// TwinCAT 3 PLC project PRG_Test_Base
// ProgramVersion: 3.1.4024.0
// libraries:
//   B_Base, * (RafalOS)
//   B_Base_HMI_Connector, * (RafalOS)
//   Tc2_Standard, * (Beckhoff Automation GmbH)
//   Tc2_System, * (Beckhoff Automation GmbH)
//   Tc3_Module, * (Beckhoff Automation GmbH)
//   TcUnit, * (www.tcunit.org)
// project tree:
//   GVLs/ GVL.TcGVL, GVL_Variable.TcGVL, GVL_VariableHMI.TcGVL
//   / PlcTask.TcTTO (not stored)
//   POUs/A0_BaseFB/Command/ FB_CommandChild.TcPOU, FB_CommandTest.TcPOU, FB_Impulstest.TcPOU (not stored)
//   POUs/A0_BaseFB/Time/ FB_BaseTimeTest.TcPOU (not stored)
//   POUs/A2_logger/ FB_LoggerTest.TcPOU
//   POUs/A4_Component/ FB_Component.TcPOU, FB_Component_HMI.TcPOU, ITF_Component.TcIO, ITF_Component_HMI.TcIO, ITF_Component_HMI_Connector.TcIO, ITF_Component_HMI_Init.TcIO (not stored), ST_Component_HMI.TcDUT, ST_Component_HMI_Link.TcDUT (not stored)
//   POUs/A5_ControlElement/ FB_ControlElement.TcPOU, FB_ControlElement_HMI.TcPOU, ITF_ControlElement.TcIO, ITF_ControlElement_HMI.TcIO, ITF_ControlElement_HMI_Connector.TcIO, ITF_ControlElement_HMI_Init.TcIO, ST_ControlElement_HMI.TcDUT, ST_ControlElement_HMI_Link.TcDUT
//   POUs/A5_ControlElement_1/ FB_ControlElement_1.TcPOU (not stored), FB_ControlElement_HMI_1.TcPOU (not stored), ITF_ControlElement_1.TcIO, ITF_ControlElement_HMI_1.TcIO (not stored), ITF_ControlElement_HMI_Connector_1.TcIO, ITF_ControlElement_HMI_Init_1.TcIO, ST_ControlElement_HMI_1.TcDUT, ST_ControlElement_HMI_Link_1.TcDUT
//   POUs/A6_GroupElement/ FB_GroupElement.TcPOU, FB_GroupElement_HMI.TcPOU, ITF_GroupElement.TcIO, ITF_GroupElement_HMI.TcIO, ITF_GroupElement_HMI_Connector.TcIO (not stored), ITF_GroupElement_HMI_Init.TcIO, ST_GroupElement_HMI.TcDUT, ST_GroupElement_HMI_Link.TcDUT
//   POUs/A7_TopElement/ FB_TopElement.TcPOU, FB_TopElement_HMI.TcPOU, ITF_TopElement.TcIO, ITF_TopElement_HMI.TcIO, ITF_TopElement_HMI_Connector.TcIO (not stored), ITF_TopElement_HMI_Init.TcIO (not stored), ST_TopElement_HMI.TcDUT, ST_TopElement_HMI_Link.TcDUT
//   POUs/A8_CommunicatorTest/ FB_CommunicatorClient.TcPOU
//   POUs/ FB_ItemTest.TcPOU
//   TESTs/ PRG_Test.TcPOU
// real-time tasks:
//   TASK PlcTask: cycle T#10ms, priority 20, ADS port 350

// ---- POUs/A4_Component/ST_Component_HMI.TcDUT
TYPE ST_Component_HMI EXTENDS ST_BaseComponent_HMI :
STRUCT
	
END_STRUCT
END_TYPE

// ---- POUs/A5_ControlElement/ST_ControlElement_HMI.TcDUT
TYPE ST_ControlElement_HMI :
STRUCT
	bZmiennaControlElement		: BOOL;
	
END_STRUCT
END_TYPE

// ---- POUs/A5_ControlElement/ST_ControlElement_HMI_Link.TcDUT
TYPE ST_ControlElement_HMI_Link EXTENDS ST_BaseControlElement_HMI_Link :
STRUCT
	stControlElement			: ST_ControlElement_HMI;
END_STRUCT
END_TYPE

// ---- POUs/A5_ControlElement_1/ST_ControlElement_HMI_1.TcDUT
TYPE ST_ControlElement_HMI_1 :
STRUCT
	bZmiennaControlElement_1		: BOOL;
	
END_STRUCT
END_TYPE

// ---- POUs/A5_ControlElement_1/ST_ControlElement_HMI_Link_1.TcDUT
TYPE ST_ControlElement_HMI_Link_1 EXTENDS ST_BaseControlElement_HMI_Link :
STRUCT
	stControlElement			: ST_ControlElement_HMI_1;
	
	stComponent1				: ST_Component_HMI_Link;
	stComponent2				: ST_Component_HMI_Link;
	
END_STRUCT
END_TYPE

// ---- POUs/A6_GroupElement/ST_GroupElement_HMI.TcDUT
TYPE ST_GroupElement_HMI :
STRUCT
	bZmiennaGroupElement	: BOOL;
	
END_STRUCT
END_TYPE

// ---- POUs/A6_GroupElement/ST_GroupElement_HMI_Link.TcDUT
TYPE ST_GroupElement_HMI_Link EXTENDS ST_BaseGroupElement_HMI_Link :
STRUCT
	stGroupElement			: ST_GroupElement_HMI;
END_STRUCT
END_TYPE

// ---- POUs/A7_TopElement/ST_TopElement_HMI.TcDUT
TYPE ST_TopElement_HMI :
STRUCT
	bZmiennaTopElement			: BOOL;
	
END_STRUCT
END_TYPE

// ---- POUs/A7_TopElement/ST_TopElement_HMI_Link.TcDUT
TYPE ST_TopElement_HMI_Link EXTENDS ST_BaseTopElement_HMI_Link :
STRUCT
	stTopElement			: ST_TopElement_HMI;

	stControlElement1		: ST_ControlElement_HMI_Link;
	stControlElement2		: ST_ControlElement_HMI_Link;
	stGroupElement1			: ST_GroupElement_HMI_Link;
	stComponent1			: ST_Component_HMI_Link;
	stComponent2			: ST_Component_HMI_Link;
	stComponent3			: ST_Component_HMI_Link;
END_STRUCT
END_TYPE

// ---- GVLs/GVL.TcGVL
{attribute 'qualified_only'}
VAR_GLOBAL
	fbMyTime				: FB_BaseTime;
	fbMyLocation			: FB_BaseLocation;
	fbLogger				: FB_BaseLogger;
	fbSS1					: FB_BaseFlag;
	fbSTO					: FB_BaseFlag;
	
	fbCommandEasy			: FB_BaseCommand;
	fbCommand				: FB_CommandChild;
	
	fbImpuls				: FB_BaseImpulse;
	
	fbCommunicator			: FB_BaseCommunicator;
	
	fbRecipe				: FB_BaseRecipe;
	fbCreatingTemplate1		: FB_CreateTepletate1;
	fbCreatingTemplate2		: FB_CreateTepletate2;
	
	stCommonData			: ST_BaseCommonData;
	
	stTopElementData		: ST_TopElement_HMI_Link;
	
	
END_VAR

// ---- GVLs/GVL_Variable.TcGVL
{attribute 'qualified_only'}
VAR_GLOBAL
	fbBasetest					: FB_Base;
	
	fbPB1_Wyk1_K1				: FB_Component;
	fbPB1_Wyk1_K2				: FB_Component;
	fbPB1_Wyk1					: FB_ControlElement (fbPB1_Wyk1_K1, fbPB1_Wyk1_K2);
	
	fbPB1_Wyk2_K1				: FB_Component;
	fbPB1_Wyk2_K2				: FB_Component;
	fbPB1_Wyk2					: FB_ControlElement_1 (fbPB1_Wyk2_K1, fbPB1_Wyk2_K2);

	fbPB1_ZL1_Wyk1_K1			: FB_Component;
	fbPB1_ZL1_Wyk1_K2			: FB_Component;
	fbPB1_ZL1_Wyk1				: FB_ControlElement (fbPB1_ZL1_Wyk1_K1, fbPB1_ZL1_Wyk1_K2);
	fbPB1_ZL1_Wyk2_K1			: FB_Component;
	fbPB1_ZL1_Wyk2_K2			: FB_Component;
	fbPB1_ZL1_Wyk2				: FB_ControlElement (fbPB1_ZL1_Wyk2_K1, fbPB1_ZL1_Wyk2_K2);
	fbPB1_ZL1_K1				: FB_Component;
	fbPB1_ZL1_K2				: FB_Component;
	fbPB1_ZL1					: FB_GroupElement (fbPB1_ZL1_Wyk1, fbPB1_ZL1_Wyk2, fbPB1_ZL1_K1, fbPB1_ZL1_K2);
	
	fbPB1_K1					: FB_Component;
	fbPB1_K2					: FB_Component;
	fbPB1_K3					: FB_Component;
	
	fbPB1						: FB_TopElement (fbPB1_Wyk1, fbPB1_Wyk2, fbPB1_ZL1, fbPB1_K1, fbPB1_K2, fbPB1_K3);
	
END_VAR

// ---- GVLs/GVL_VariableHMI.TcGVL
{attribute 'qualified_only'}
VAR_GLOBAL
//	fbComponentHMI_1			: FB_Component_HMI (itfBaseLoggerConnector := GVL.fbLogger, itfComponentConnector := GVL_Variable.fbComponent_1);
//	fbControlrElementHMI_1		: FB_ControlElement_HMI (itfBaseLoggerConnector := GVL.fbLogger, itfControlElementConnector := GVL_Variable.fbControlElement_1);
//	fbGroupElementHMI_1			: FB_GroupElement_HMI (itfBaseLoggerConnector := GVL.fbLogger, itfGroupelementConnector := GVL_Variable.fbGroupElement_1);
//	fbTopElementHMI_1			: FB_TopElement_HMI (itfBaseLoggerConnector := GVL.fbLogger, itfTopElementConnector := GVL_Variable.fbTopElement_1);
//
//	fbComponentHMI_1_L			: FB_Component_HMI (itfBaseLoggerConnector := GVL.fbLogger, itfComponentConnector := GVL_Variable.fbComponent_1_L);
//	fbComponentHMI_2_L			: FB_Component_HMI (itfBaseLoggerConnector := GVL.fbLogger, itfComponentConnector := GVL_Variable.fbComponent_2_L);
//	fbComponentHMI_3_L			: FB_Component_HMI (itfBaseLoggerConnector := GVL.fbLogger, itfComponentConnector := GVL_Variable.fbComponent_3_L);

	
END_VAR

// ---- POUs/A4_Component/ITF_Component.TcIO
INTERFACE ITF_Component EXTENDS ITF_BaseComponent

END_INTERFACE

// ---- POUs/A4_Component/ITF_Component_HMI.TcIO
INTERFACE ITF_Component_HMI

METHOD LinkComponentData : BOOL
VAR_INPUT
	stData					: REFERENCE TO ST_Component_HMI_Link;
END_VAR
END_METHOD

END_INTERFACE

// ---- POUs/A4_Component/ITF_Component_HMI_Connector.TcIO
INTERFACE ITF_Component_HMI_Connector EXTENDS ITF_BaseComponent_HMI_Connector

END_INTERFACE

// ---- POUs/A5_ControlElement/ITF_ControlElement.TcIO
INTERFACE ITF_ControlElement

END_INTERFACE

// ---- POUs/A5_ControlElement/ITF_ControlElement_HMI.TcIO
INTERFACE ITF_ControlElement_HMI EXTENDS ITF_BaseComponent_HMI

METHOD LinkControlElementData : BOOL
VAR_INPUT
	stData				: REFERENCE TO ST_ControlElement_HMI_Link;
END_VAR
END_METHOD

END_INTERFACE

// ---- POUs/A5_ControlElement/ITF_ControlElement_HMI_Connector.TcIO
INTERFACE ITF_ControlElement_HMI_Connector EXTENDS ITF_BaseControlElement_HMI_Connector

END_INTERFACE

// ---- POUs/A5_ControlElement/ITF_ControlElement_HMI_Init.TcIO
INTERFACE ITF_ControlElement_HMI_Init EXTENDS ITF_BaseControlElement, ITF_ControlElement_HMI_Connector

END_INTERFACE

// ---- POUs/A5_ControlElement_1/ITF_ControlElement_1.TcIO
INTERFACE ITF_ControlElement_1 EXTENDS ITF_BaseControlElement

END_INTERFACE

// ---- POUs/A5_ControlElement_1/ITF_ControlElement_HMI_Connector_1.TcIO
INTERFACE ITF_ControlElement_HMI_Connector_1 EXTENDS ITF_BaseControlElement_HMI_Connector

END_INTERFACE

// ---- POUs/A5_ControlElement_1/ITF_ControlElement_HMI_Init_1.TcIO
INTERFACE ITF_ControlElement_HMI_Init_1 EXTENDS ITF_BaseControlElement, ITF_ControlElement_HMI_Connector_1

END_INTERFACE

// ---- POUs/A6_GroupElement/ITF_GroupElement.TcIO
INTERFACE ITF_GroupElement EXTENDS ITF_BaseGroupElement

END_INTERFACE

// ---- POUs/A6_GroupElement/ITF_GroupElement_HMI.TcIO
INTERFACE ITF_GroupElement_HMI EXTENDS ITF_BaseGroupElement_HMI

METHOD LinkGroupelementData : BOOL
VAR_INPUT
	stData					: REFERENCE TO ST_GroupElement_HMI_Link;
END_VAR
END_METHOD

END_INTERFACE

// ---- POUs/A6_GroupElement/ITF_GroupElement_HMI_Init.TcIO
INTERFACE ITF_GroupElement_HMI_Init EXTENDS ITF_BaseGroupElement, ITF_GroupElement_HMI_Connector

END_INTERFACE

// ---- POUs/A7_TopElement/ITF_TopElement.TcIO
INTERFACE ITF_TopElement EXTENDS ITF_BaseTopElement

END_INTERFACE

// ---- POUs/A7_TopElement/ITF_TopElement_HMI.TcIO
INTERFACE ITF_TopElement_HMI

METHOD LinkTopElementData : BOOL
VAR_INPUT
	stData				: REFERENCE TO ST_TopElement_HMI_Link;
END_VAR
END_METHOD

END_INTERFACE

// ---- POUs/A0_BaseFB/Command/FB_CommandChild.TcPOU
FUNCTION_BLOCK FB_CommandChild EXTENDS FB_BaseCommand
VAR
	bFinish				: BOOL;
	iI1					: INT;
	iI2					: INT;
END_VAR

IF (THIS^.GetFirstCycle ()) THEN
	iI1 := iI1 + 1;
END_IF
IF (THIS^.GetLastCycle ()) THEN
	iI2 := iI2 + 1;
END_IF

METHOD PUBLIC CyklTestu : BOOL
VAR_INPUT
END_VAR
CASE THIS^.GetStep () OF
0	:
	THIS^.SetStepINC10 ();
10	:
	IF (THIS^.bFinish) THEN
		THIS^.SetStepAsFinal ();
	END_IF
END_CASE
CyklTestu			:= THIS^.TestingLastCycle ();
END_METHOD

END_FUNCTION_BLOCK

// ---- POUs/A4_Component/FB_Component.TcPOU
FUNCTION_BLOCK FB_Component EXTENDS FB_BaseComponent IMPLEMENTS ITF_Component, ITF_Component_HMI_Init
VAR
	bSetAlarm		: BOOL;
	bSetError1		: BOOL;
	bSetError2		: BOOL;
	sttmpEvent		: ST_BaseEvents_RowInQueue;
END_VAR

IF (bSetAlarm) THEN
	bSetAlarm		:= FALSE;
	
END_IF
IF (bSetError1) THEN
	bSetError1		:= FALSE;
	
END_IF
IF (bSetError2) THEN
	bSetError2		:= FALSE;
	
END_IF

(*			
	EVERDE sp. z o.o.
	Rafał Osajda		24.03.2025		TC 4024.66
	Definicja nowego zgłoszenia
*)
METHOD PUBLIC EventsDefinition : BOOL
VAR
	fbName					: FB_BaseLabel;
END_VAR
SUPER^.EventsDefinition ();

fbName.SetText (eLocation := E_BaseLocation.pl, wsDescription := "Zgloszneie komponentu 1 PL");
fbName.SetText (eLocation := E_BaseLocation.en, wsDescription := "Zgloszneie komponentu 1 EN");
fbName.SetText (eLocation := E_BaseLocation.de, wsDescription := "Zgloszneie komponentu 1 DE");
THIS^.AddEvent (
	bIgnoreRepetitions		:= TRUE,
	eEventCategory			:= E_BaseEvents_Category.ALARM,
	bConfirm				:= FALSE,
	stDescription			:= fbName.GetTexts ()
);

fbName.SetText (eLocation := E_BaseLocation.pl, wsDescription := "Zgloszneie komponentu 2 PL");
fbName.SetText (eLocation := E_BaseLocation.en, wsDescription := "Zgloszneie komponentu 2 EN");
fbName.SetText (eLocation := E_BaseLocation.de, wsDescription := "Zgloszneie komponentu 2 DE");
THIS^.AddEvent (
	bIgnoreRepetitions		:= TRUE,
	eEventCategory			:= E_BaseEvents_Category.Error,
	bConfirm				:= FALSE,
	stDescription			:= fbName.GetTexts ()
);

fbName.SetText (eLocation := E_BaseLocation.pl, wsDescription := "Zgloszneie komponentu 3 PL");
fbName.SetText (eLocation := E_BaseLocation.en, wsDescription := "Zgloszneie komponentu 3 EN");
fbName.SetText (eLocation := E_BaseLocation.de, wsDescription := "Zgloszneie komponentu 3 DE");
THIS^.AddEvent (
	bIgnoreRepetitions		:= TRUE,
	eEventCategory			:= E_BaseEvents_Category.Error,
	bConfirm				:= TRUE,
	stDescription			:= fbName.GetTexts ()
);
END_METHOD

END_FUNCTION_BLOCK

// ---- POUs/A5_ControlElement/FB_ControlElement.TcPOU
FUNCTION_BLOCK FB_ControlElement EXTENDS FB_BaseControlElement IMPLEMENTS ITF_ControlElement, ITF_ControlElement_HMI_Init
VAR
	itfComponent1				: ITF_Component;
	itfComponent2				: ITF_Component;
END_VAR

(*			
	EVERDE sp. z o.o.
	Rafał Osajda		24.03.2025		TC 4024.66
	Definicja nowego zgłoszenia
*)
METHOD PUBLIC EventsDefinition : BOOL
VAR
	fbName					: FB_BaseLabel;
END_VAR
SUPER^.EventsDefinition ();

fbName.SetText (eLocation := E_BaseLocation.pl, wsDescription := "Zgloszneie Wykonawczego 1 PL");
fbName.SetText (eLocation := E_BaseLocation.en, wsDescription := "Zgloszneie Wykonawczego 1 EN");
fbName.SetText (eLocation := E_BaseLocation.de, wsDescription := "Zgloszneie Wykonawczego 1 DE");
THIS^.AddEvent (
	bIgnoreRepetitions		:= TRUE,
	eEventCategory			:= E_BaseEvents_Category.ALARM,
	bConfirm				:= FALSE,
	stDescription			:= fbName.GetTexts ()
);

fbName.SetText (eLocation := E_BaseLocation.pl, wsDescription := "Zgloszneie Wykonawczego 2 PL");
fbName.SetText (eLocation := E_BaseLocation.en, wsDescription := "Zgloszneie Wykonawczego 2 EN");
fbName.SetText (eLocation := E_BaseLocation.de, wsDescription := "Zgloszneie Wykonawczego 2 DE");
THIS^.AddEvent (
	bIgnoreRepetitions		:= TRUE,
	eEventCategory			:= E_BaseEvents_Category.ALARM,
	bConfirm				:= FALSE,
	stDescription			:= fbName.GetTexts ()
);

fbName.SetText (eLocation := E_BaseLocation.pl, wsDescription := "Zgloszneie Wykonawczego 3 PL");
fbName.SetText (eLocation := E_BaseLocation.en, wsDescription := "Zgloszneie Wykonawczego 3 EN");
fbName.SetText (eLocation := E_BaseLocation.de, wsDescription := "Zgloszneie Wykonawczego 3 DE");
THIS^.AddEvent (
	bIgnoreRepetitions		:= TRUE,
	eEventCategory			:= E_BaseEvents_Category.ALARM,
	bConfirm				:= FALSE,
	stDescription			:= fbName.GetTexts ()
);
END_METHOD

METHOD FB_init : BOOL
VAR_INPUT
	bInitRetains : BOOL; // if TRUE, the retain variables are initialized (warm start / cold start)
	bInCopyCode : BOOL;  // if TRUE, the instance afterwards gets moved into the copy code (online change)
	itfComponent1				: ITF_Component;
	itfComponent2				: ITF_Component;
END_VAR
THIS^.itfComponent1					:= itfComponent1;
THIS^.AddComponent (itfComponent	:= itfComponent1);
THIS^.SetText (eLocation 			:= E_BaseLocation.pl, wsDescription := "Nazwa komponentu 1 pl");
THIS^.SetText (eLocation 			:= E_BaseLocation.en, wsDescription := "Nazwa komponentu 1 en");
THIS^.SetText (eLocation 			:= E_BaseLocation.de, wsDescription := "Nazwa komponentu 1 de");
THIS^.itfComponent1.SetName (stName	:= THIS^.GetTexts ());

THIS^.itfComponent2					:= itfComponent2;
THIS^.AddComponent (itfComponent	:= itfComponent2);
THIS^.SetText (eLocation 			:= E_BaseLocation.pl, wsDescription := "Nazwa komponentu 2 pl");
THIS^.SetText (eLocation 			:= E_BaseLocation.en, wsDescription := "Nazwa komponentu 2 en");
THIS^.SetText (eLocation 			:= E_BaseLocation.de, wsDescription := "Nazwa komponentu 2 de");
THIS^.itfComponent2.SetName (stName	:= THIS^.GetTexts ());
END_METHOD

END_FUNCTION_BLOCK

// ---- POUs/A6_GroupElement/FB_GroupElement.TcPOU
FUNCTION_BLOCK FB_GroupElement EXTENDS FB_BaseGroupElement IMPLEMENTS ITF_GroupElement, ITF_GroupElement_HMI_Init
VAR
	itfControlElement1			: ITF_ControlElement;
	itfControlElement2			: ITF_ControlElement;
	itfComponent1				: ITF_Component;
	itfComponent2				: ITF_Component;
END_VAR

(*			
	EVERDE sp. z o.o.
	Rafał Osajda		24.03.2025		TC 4024.66
	Definicja nowego zgłoszenia
*)
METHOD PUBLIC EventsDefinition : BOOL
VAR
	fbName					: FB_BaseLabel;
END_VAR
SUPER^.EventsDefinition ();

fbName.SetText (eLocation := E_BaseLocation.pl, wsDescription := "Zgloszneie Zlozonego 1 PL");
fbName.SetText (eLocation := E_BaseLocation.en, wsDescription := "Zgloszneie Zlozonego 1 EN");
fbName.SetText (eLocation := E_BaseLocation.de, wsDescription := "Zgloszneie Zlozonego 1 DE");
THIS^.AddEvent (
	bIgnoreRepetitions		:= TRUE,
	eEventCategory			:= E_BaseEvents_Category.ALARM,
	bConfirm				:= FALSE,
	stDescription			:= fbName.GetTexts ()
);

fbName.SetText (eLocation := E_BaseLocation.pl, wsDescription := "Zgloszneie Zlozonego 2 PL");
fbName.SetText (eLocation := E_BaseLocation.en, wsDescription := "Zgloszneie Zlozonego 2 EN");
fbName.SetText (eLocation := E_BaseLocation.de, wsDescription := "Zgloszneie Zlozonego 2 DE");
THIS^.AddEvent (
	bIgnoreRepetitions		:= TRUE,
	eEventCategory			:= E_BaseEvents_Category.ALARM,
	bConfirm				:= FALSE,
	stDescription			:= fbName.GetTexts ()
);

fbName.SetText (eLocation := E_BaseLocation.pl, wsDescription := "Zgloszneie Zlozonego 3 PL");
fbName.SetText (eLocation := E_BaseLocation.en, wsDescription := "Zgloszneie Zlozonego 3 EN");
fbName.SetText (eLocation := E_BaseLocation.de, wsDescription := "Zgloszneie Zlozonego 3 DE");
THIS^.AddEvent (
	bIgnoreRepetitions		:= TRUE,
	eEventCategory			:= E_BaseEvents_Category.ALARM,
	bConfirm				:= FALSE,
	stDescription			:= fbName.GetTexts ()
);
END_METHOD

METHOD FB_init : BOOL
VAR_INPUT
	bInitRetains : BOOL; // if TRUE, the retain variables are initialized (warm start / cold start)
	bInCopyCode : BOOL;  // if TRUE, the instance afterwards gets moved into the copy code (online change)
	itfControlElement1			: ITF_ControlElement;
	itfControlElement2			: ITF_ControlElement;
	itfComponent1				: ITF_Component;
	itfComponent2				: ITF_Component;
END_VAR
THIS^.itfControlElement1			:= itfControlElement1;
THIS^.AddControlElement (itfControlElement	:= itfControlElement1);
THIS^.SetText (eLocation 			:= E_BaseLocation.pl, wsDescription := "Nazwa komponentu zlozenia 1 pl");
THIS^.SetText (eLocation 			:= E_BaseLocation.pl, wsDescription := "Nazwa komponentu zlozenia 1 en");
THIS^.SetText (eLocation 			:= E_BaseLocation.pl, wsDescription := "Nazwa komponentu zlozenia 1 de");
THIS^.itfControlElement1.SetName (stName	:= THIS^.GetTexts ());

THIS^.itfControlElement2			:= itfControlElement2;
THIS^.AddControlElement (itfControlElement	:= itfControlElement2);
THIS^.SetText (eLocation 			:= E_BaseLocation.pl, wsDescription := "Nazwa komponentu zlozenia 1 pl");
THIS^.SetText (eLocation 			:= E_BaseLocation.en, wsDescription := "Nazwa komponentu zlozenia 1 en");
THIS^.SetText (eLocation 			:= E_BaseLocation.de, wsDescription := "Nazwa komponentu zlozenia 1 de");
THIS^.itfControlElement2.SetName (stName	:= THIS^.GetTexts ());

THIS^.itfComponent1					:= itfComponent1;
THIS^.AddComponent (itfComponent	:= itfComponent1);
THIS^.SetText (eLocation 			:= E_BaseLocation.pl, wsDescription := "Nazwa komponentu zlozenia 1 pl");
THIS^.SetText (eLocation 			:= E_BaseLocation.en, wsDescription := "Nazwa komponentu zlozenia 1 en");
THIS^.SetText (eLocation 			:= E_BaseLocation.de, wsDescription := "Nazwa komponentu zlozenia 1 de");
THIS^.itfComponent1.SetName (stName	:= THIS^.GetTexts ());

THIS^.itfComponent2					:= itfComponent2;
THIS^.AddComponent (itfComponent	:= itfComponent2);
THIS^.SetText (eLocation 			:= E_BaseLocation.pl, wsDescription := "Nazwa komponentu złożenia 2 pl");
THIS^.SetText (eLocation 			:= E_BaseLocation.en, wsDescription := "Nazwa komponentu złożenia 2 en");
THIS^.SetText (eLocation 			:= E_BaseLocation.de, wsDescription := "Nazwa komponentu złożenia 2 de");
THIS^.itfComponent2.SetName (stName	:= THIS^.GetTexts ());
END_METHOD

END_FUNCTION_BLOCK

// ---- POUs/A7_TopElement/FB_TopElement.TcPOU
FUNCTION_BLOCK FB_TopElement EXTENDS FB_BaseTopElement IMPLEMENTS ITF_TopElement, ITF_TopElement_HMI_Init
VAR
	itfControlElement1				: ITF_ControlElement;
	itfControlElement2				: ITF_ControlElement_1;
	itfGroupElement1				: ITF_GroupElement;
	itfComponent1					: ITF_Component;
	itfComponent2					: ITF_Component;
	itfComponent3					: ITF_Component;
END_VAR

(*			
	EVERDE sp. z o.o.
	Rafał Osajda		24.03.2025		TC 4024.66
	Definicja nowego zgłoszenia
*)
METHOD PUBLIC EventsDefinition : BOOL
VAR
	fbName					: FB_BaseLabel;
END_VAR
SUPER^.EventsDefinition ();

fbName.SetText (eLocation := E_BaseLocation.pl, wsDescription := "Zgloszneie PB 1 PL");
fbName.SetText (eLocation := E_BaseLocation.en, wsDescription := "Zgloszneie PB 1 EN");
fbName.SetText (eLocation := E_BaseLocation.de, wsDescription := "Zgloszneie PB 1 DE");
THIS^.AddEvent (
	bIgnoreRepetitions		:= TRUE,
	eEventCategory			:= E_BaseEvents_Category.ALARM,
	bConfirm				:= FALSE,
	stDescription			:= fbName.GetTexts ()
);

fbName.SetText (eLocation := E_BaseLocation.pl, wsDescription := "Zgloszneie PB 2 PL");
fbName.SetText (eLocation := E_BaseLocation.en, wsDescription := "Zgloszneie PB 2 EN");
fbName.SetText (eLocation := E_BaseLocation.de, wsDescription := "Zgloszneie PB 2 DE");
THIS^.AddEvent (
	bIgnoreRepetitions		:= TRUE,
	eEventCategory			:= E_BaseEvents_Category.ALARM,
	bConfirm				:= FALSE,
	stDescription			:= fbName.GetTexts ()
);

fbName.SetText (eLocation := E_BaseLocation.pl, wsDescription := "Zgloszneie PB 3 PL");
fbName.SetText (eLocation := E_BaseLocation.en, wsDescription := "Zgloszneie PB 3 EN");
fbName.SetText (eLocation := E_BaseLocation.de, wsDescription := "Zgloszneie PB 3 DE");
THIS^.AddEvent (
	bIgnoreRepetitions		:= TRUE,
	eEventCategory			:= E_BaseEvents_Category.ALARM,
	bConfirm				:= FALSE,
	stDescription			:= fbName.GetTexts ()
);
END_METHOD

METHOD FB_init : BOOL
VAR_INPUT
	bInitRetains : BOOL; // if TRUE, the retain variables are initialized (warm start / cold start)
	bInCopyCode : BOOL;  // if TRUE, the instance afterwards gets moved into the copy code (online change)
	itfControlElement1				: ITF_ControlElement;
	itfControlElement2				: ITF_ControlElement_1;
	itfGroupElement1				: ITF_GroupElement;
	itfComponent1					: ITF_Component;
	itfComponent2					: ITF_Component;
	itfComponent3					: ITF_Component;
END_VAR
THIS^.itfControlElement1			:= itfControlElement1;
THIS^.AddControlElement (itfControlElement	:= itfControlElement1);
THIS^.SetText (eLocation 			:= E_BaseLocation.pl, wsDescription := "Nazwa control eleemntu PB - 1");
THIS^.SetText (eLocation 			:= E_BaseLocation.pl, wsDescription := "Nazwa control eleemntu PB - 1");
THIS^.SetText (eLocation 			:= E_BaseLocation.pl, wsDescription := "Nazwa control eleemntu PB - 1");
THIS^.itfControlElement1.SetName (stName	:= THIS^.GetTexts ());

THIS^.itfControlElement2			:= itfControlElement2;
THIS^.AddControlElement (itfControlElement	:= itfControlElement2);
THIS^.SetText (eLocation 			:= E_BaseLocation.pl, wsDescription := "Nazwa control elementu PB - 2");
THIS^.SetText (eLocation 			:= E_BaseLocation.pl, wsDescription := "Nazwa control elementu PB - 2");
THIS^.SetText (eLocation 			:= E_BaseLocation.pl, wsDescription := "Nazwa control elementu PB - 2");
THIS^.itfControlElement2.SetName (stName	:= THIS^.GetTexts ());

THIS^.itfGroupElement1				:= itfGroupElement1;
THIS^.AddControlElement (itfControlElement	:= itfGroupElement1);
THIS^.SetText (eLocation 			:= E_BaseLocation.pl, wsDescription := "Nazwa group elementu PB - 1");
THIS^.SetText (eLocation 			:= E_BaseLocation.pl, wsDescription := "Nazwa group elementu PB - 1");
THIS^.SetText (eLocation 			:= E_BaseLocation.pl, wsDescription := "Nazwa group elementu PB - 1");
THIS^.itfGroupElement1.SetName (stName	:= THIS^.GetTexts ());

THIS^.itfComponent1					:= itfComponent1;
THIS^.AddComponent (itfComponent	:= itfComponent1);
THIS^.SetText (eLocation 			:= E_BaseLocation.pl, wsDescription := "Nazwa komponentu PB - 1");
THIS^.SetText (eLocation 			:= E_BaseLocation.pl, wsDescription := "Nazwa komponentu PB - 1");
THIS^.SetText (eLocation 			:= E_BaseLocation.pl, wsDescription := "Nazwa komponentu PB - 1");
THIS^.itfComponent1.SetName (stName	:= THIS^.GetTexts ());

THIS^.itfComponent2					:= itfComponent2;
THIS^.AddComponent (itfComponent	:= itfComponent2);
THIS^.SetText (eLocation 			:= E_BaseLocation.pl, wsDescription := "Nazwa komponentu PB -2");
THIS^.SetText (eLocation 			:= E_BaseLocation.pl, wsDescription := "Nazwa komponentu PB -2");
THIS^.SetText (eLocation 			:= E_BaseLocation.pl, wsDescription := "Nazwa komponentu PB -2");
THIS^.itfComponent2.SetName (stName	:= THIS^.GetTexts ());

THIS^.itfComponent3					:= itfComponent3;
THIS^.AddComponent (itfComponent	:= itfComponent3);
THIS^.SetText (eLocation 			:= E_BaseLocation.pl, wsDescription := "Nazwa komponentu PB - 3");
THIS^.SetText (eLocation 			:= E_BaseLocation.pl, wsDescription := "Nazwa komponentu PB - 3");
THIS^.SetText (eLocation 			:= E_BaseLocation.pl, wsDescription := "Nazwa komponentu PB - 3");
THIS^.itfComponent3.SetName (stName	:= THIS^.GetTexts ());
END_METHOD

END_FUNCTION_BLOCK

// ---- POUs/A4_Component/FB_Component_HMI.TcPOU
FUNCTION_BLOCK FB_Component_HMI EXTENDS FB_BaseComponent_HMI IMPLEMENTS ITF_Component_HMI
VAR
	itfComponentConnector				: ITF_Component_HMI_Connector;
	refstComponentData					: REFERENCE TO ST_Component_HMI;
	
END_VAR

METHOD FB_init : BOOL
VAR_INPUT
	bInitRetains : BOOL; // if TRUE, the retain variables are initialized (warm start / cold start)
	bInCopyCode : BOOL;  // if TRUE, the instance afterwards gets moved into the copy code (online change)
	itfBaseLoggerConnector				: ITF_BaseLogger_HMI_Connector;	//bezpośredni łącznik do logera
	itfComponentConnector				: ITF_Component_HMI_Init;
END_VAR
//Przypisanie do elementu który własnie stworzyliśmy
THIS^.itfComponentConnector				:= itfComponentConnector;
//Przypisanie do elementów z biblioteki
THIS^.itfBaseLoggerElementConnector		:= itfComponentConnector;
THIS^.itfBaseComponentConnector			:= itfComponentConnector;

//
THIS^.itfBaseLoggerConnector			:= itfBaseLoggerConnector;

IF (THIS^.itfComponentConnector <> 0 AND
	THIS^.itfBaseLoggerElementConnector <> 0 AND
	THIS^.itfBaseComponentConnector	<> 0 AND
	THIS^.itfBaseLoggerConnector <> 0) THEN
	THIS^.bIsInit						:= TRUE;
END_IF
END_METHOD

METHOD LinkComponentData : BOOL
VAR_INPUT
	stData					: REFERENCE TO ST_Component_HMI_Link;
END_VAR
THIS^.refstComponentData	REF= stData.stComponent;

THIS^.refstBaseLoggerElementDataHMI	REF= stData.stBaseLoggerElement;
THIS^.refstBaseComponentDataHMI		REF= stData.stBaseComponent;

THIS^.CreateLinkToEventsMemory ();

IF (__ISVALIDREF (THIS^.refstComponentData) AND
	__ISVALIDREF (THIS^.refstBaseLoggerElementDataHMI) AND
	__ISVALIDREF (THIS^.refstBaseComponentDataHMI) ) THEN
	THIS^.bIsValidData		:= TRUE;
	LinkComponentData		:= TRUE;
END_IF
END_METHOD

END_FUNCTION_BLOCK

// ---- POUs/A5_ControlElement/FB_ControlElement_HMI.TcPOU
FUNCTION_BLOCK FB_ControlElement_HMI EXTENDS FB_BaseControlElement_HMI IMPLEMENTS ITF_ControlElement_HMI
VAR
	itfControlElementConnector			: ITF_ControlElement_HMI_Connector;
	refstControlElementData				: REFERENCE TO ST_ControlElement_HMI;
	
	itfComponent1						: ITF_Component_HMI;
	itfComponent2						: ITF_Component_HMI;
END_VAR

METHOD FB_init : BOOL
VAR_INPUT
	bInitRetains : BOOL; // if TRUE, the retain variables are initialized (warm start / cold start)
	bInCopyCode : BOOL;  // if TRUE, the instance afterwards gets moved into the copy code (online change)
	itfBaseLoggerConnector				: ITF_BaseLogger_HMI_Connector;	//bezpośredni łącznik do logera
	itfControlElementConnector			: ITF_ControlElement_HMI_Init;
	itfComponent1						: ITF_Component_HMI;
	itfComponent2						: ITF_Component_HMI;
END_VAR
//Przypisanie do elementu który własnie stworzyliśmy
THIS^.itfControlElementConnector		:= itfControlElementConnector;
//Przypisanie do elementów z biblioteki
THIS^.itfBaseLoggerElementConnector		:= itfControlElementConnector;
THIS^.itfBaseComponentConnector			:= itfControlElementConnector;
THIS^.itfBaseControlElementConnector	:= itfControlElementConnector;
//
THIS^.itfBaseLoggerConnector			:= itfBaseLoggerConnector;
//
THIS^.itfComponent1						:= itfComponent1;
THIS^.AddComponent (itfComponentHMI		:= itfComponent1);
THIS^.itfComponent2						:= itfComponent2;
this^.AddComponent (itfComponentHMI		:= itfComponent2);

IF (THIS^.itfControlElementConnector <> 0 AND
	THIS^.itfBaseLoggerElementConnector <> 0 AND
	THIS^.itfBaseComponentConnector	<> 0 AND
	THIS^.itfBaseControlElementConnector <> 0 AND
	THIS^.itfBaseLoggerConnector <> 0) THEN
	THIS^.bIsInit						:= TRUE;
END_IF
END_METHOD

METHOD LinkControlElementData : BOOL
VAR_INPUT
	stData				: reference to ST_ControlElement_HMI_Link;
END_VAR
THIS^.refstControlElementData			REF= stData.stControlElement;	//ta zmienna powstaje w elemencie 

THIS^.refstBaseLoggerElementDataHMI		REF= stData.stBaseLoggerElement;	//zmienne z biblioteki ale dopiero tu je moge przypisać 
THIS^.refstBaseComponentDataHMI			REF= stData.stBaseComponent;
THIS^.refstBaseControlElementDataHMI	REF= stData.stBaseControlElement;

THIS^.itfComponent1.LinkComponentData (stData := stData.stComponent1);	//przekazanie danych do elementu podrzędnego np do czujnika
THIS^.itfComponent2.LinkComponentData (stData := stData.stComponent2);

THIS^.CreateLinkToEventsMemory ();	//wywołanie metody linkującą poamięc zgłoszęń

IF (__ISVALIDREF (THIS^.refstControlElementData) AND
	__ISVALIDREF (THIS^.refstBaseLoggerElementDataHMI) AND
	__ISVALIDREF (THIS^.refstBaseComponentDataHMI) AND
	__ISVALIDREF (THIS^.refstBaseControlElementDataHMI)) THEN
	THIS^.bIsValidData		:= TRUE;
	LinkControlElementData	:= TRUE;
END_IF
END_METHOD

END_FUNCTION_BLOCK

// ---- POUs/A6_GroupElement/FB_GroupElement_HMI.TcPOU
FUNCTION_BLOCK FB_GroupElement_HMI EXTENDS FB_BaseGroupElement_HMI IMPLEMENTS ITF_GroupElement_HMI
VAR
	itfGroupElementConnector			: ITF_GroupElement_HMI_Connector;
	refstGroupElementData				: REFERENCE TO ST_GroupElement_HMI;
	
	itfControlElement1					: ITF_ControlElement_HMI;
	itfControlElement2					: ITF_ControlElement_HMI;
	itfComponent1						: ITF_Component_HMI;
	itfComponent2						: ITF_Component_HMI;
	
END_VAR

METHOD FB_init : BOOL
VAR_INPUT
	bInitRetains : BOOL; // if TRUE, the retain variables are initialized (warm start / cold start)
	bInCopyCode : BOOL;  // if TRUE, the instance afterwards gets moved into the copy code (online change)
	itfBaseLoggerConnector				: ITF_BaseLogger_HMI_Connector;	//bezpośredni łącznik do logera
	itfGroupElementConnector			: ITF_GroupElement_HMI_Init;
	itfControlElement1					: ITF_ControlElement_HMI;
	itfControlElement2					: ITF_ControlElement_HMI;
	itfComponent1						: ITF_Component_HMI;
	itfComponent2						: ITF_Component_HMI;
	
END_VAR
//Przypisanie do elementu który własnie stworzyliśmy
THIS^.itfGroupElementConnector			:= itfGroupElementConnector;
//Przypisanie do elementów z biblioteki
THIS^.itfBaseLoggerElementConnector		:= itfGroupElementConnector;
THIS^.itfBaseComponentConnector			:= itfGroupElementConnector;
THIS^.itfBaseControlElementConnector	:= itfGroupElementConnector;
THIS^.itfBaseGroupElementConnector		:= itfGroupElementConnector;
//
THIS^.itfBaseLoggerConnector			:= itfBaseLoggerConnector;
//
THIS^.itfControlElement1				:= itfControlElement1;
THIS^.AddControlElement (itfControlElementHMI	:= itfControlElement1);
THIS^.itfControlElement2				:= itfControlElement2;
THIS^.AddControlElement (itfControlElementHMI	:= itfControlElement2);
THIS^.itfComponent1						:= itfComponent1;
THIS^.AddComponent (itfComponentHMI		:= itfComponent1);
THIS^.itfComponent2						:= itfComponent2;
THIS^.AddComponent (itfComponentHMI 	:= itfComponent2);

IF (THIS^.itfGroupElementConnector <> 0 AND
	THIS^.itfBaseLoggerElementConnector <> 0 AND
	THIS^.itfBaseComponentConnector	<> 0 AND
	THIS^.itfBaseControlElementConnector <> 0 AND
	THIS^.itfBaseGroupElementConnector <> 0 AND
	THIS^.itfBaseLoggerConnector <> 0) THEN
	THIS^.bIsInit						:= TRUE;
END_IF
END_METHOD

METHOD LinkGroupelementData : BOOL
VAR_INPUT
	stData					: REFERENCE TO ST_GroupElement_HMI_Link;
END_VAR
THIS^.refstGroupElementData	REF= stData.stGroupElement;

THIS^.refstBaseLoggerElementDataHMI	REF= stData.stBaseLoggerElement;
THIS^.refstBaseComponentDataHMI		REF= stData.stBaseComponent;
THIS^.refstBaseControlElementDataHMI	REF= stData.stBaseControlElement;
THIS^.refstBaseGroupElementDataHMI		REF= stData.stBaseGroupElement;

THIS^.itfControlElement1.LinkControlElementData (stData := stData.stControlElement1);
THIS^.itfControlElement2.LinkControlElementData (stData := stData.stControlElement2);
THIS^.itfComponent1.LinkComponentData (stData := stData.stComponent1);
THIS^.itfComponent2.LinkComponentData (stData := stData.stComponent2);

THIS^.CreateLinkToEventsMemory ();

IF (__ISVALIDREF (THIS^.refstGroupElementData) AND this^.IsLinkedReferences ()) THEN
	THIS^.bIsValidData		:= TRUE;
	LinkGroupelementData	:= TRUE;
END_IF
END_METHOD

END_FUNCTION_BLOCK

// ---- POUs/A7_TopElement/FB_TopElement_HMI.TcPOU
FUNCTION_BLOCK FB_TopElement_HMI EXTENDS FB_BaseTopElement_HMI IMPLEMENTS ITF_TopElement_HMI
VAR
	itfTopElementConnector				: ITF_TopElement_HMI_Connector;
	refstTopElementData					: REFERENCE TO ST_TopElement_HMI;
	itfControlElement1					: ITF_ControlElement_HMI;
	itfControlElement2					: ITF_ControlElement_HMI;
	itfGroupElement1					: ITF_GroupElement_HMI;
	itfComponent1						: ITF_Component_HMI;
	itfComponent2						: ITF_Component_HMI;
	itfComponent3						: ITF_Component_HMI;
END_VAR

METHOD FB_init : BOOL
VAR_INPUT
	bInitRetains : BOOL; // if TRUE, the retain variables are initialized (warm start / cold start)
	bInCopyCode : BOOL;  // if TRUE, the instance afterwards gets moved into the copy code (online change)
	itfBaseLoggerConnector				: ITF_BaseLogger_HMI_Connector;	//bezpośredni łącznik do logera
	itfTopElementConnector				: ITF_TopElement_HMI_Init;
	itfControlElement1					: ITF_ControlElement_HMI;
	itfControlElement2					: ITF_ControlElement_HMI;
	itfGroupElement1					: ITF_GroupElement_HMI;
	itfComponent1						: ITF_Component_HMI;
	itfComponent2						: ITF_Component_HMI;
	itfComponent3						: ITF_Component_HMI;
END_VAR
//Przypisanie do elementu który własnie stworzyliśmy
THIS^.itfTopElementConnector			:= itfTopElementConnector;
//Przypisanie do elementów z biblioteki
THIS^.itfBaseLoggerElementConnector		:= itfTopElementConnector;
THIS^.itfBaseComponentConnector			:= itfTopElementConnector;
THIS^.itfBaseControlElementConnector	:= itfTopElementConnector;
THIS^.itfBaseGroupElementConnector		:= itfTopElementConnector;
THIS^.itfBaseTopElementConnector		:= itfTopElementConnector;
//
THIS^.itfBaseLoggerConnector			:= itfBaseLoggerConnector;

THIS^.itfControlElement1				:= itfControlElement1;
THIS^.AddControlElement (itfControlElementHMI	:= itfControlElement1);
THIS^.itfControlElement2				:= itfControlElement2;
THIS^.AddControlElement (itfControlElementHMI	:= itfControlElement2);
THIS^.itfGroupElement1					:= itfGroupElement1;
THIS^.AddControlElement (itfControlElementHMI	:= itfGroupElement1);
THIS^.itfComponent1						:= itfComponent1;
THIS^.AddComponent (itfComponentHMI		:= itfComponent1);
THIS^.itfComponent2						:= itfComponent2;
THIS^.AddComponent (itfComponentHMI		:= itfComponent2);
THIS^.itfComponent3						:= itfComponent3;
THIS^.AddComponent (itfComponentHMI		:= itfComponent3);


IF (THIS^.itfTopElementConnector <> 0 AND
	THIS^.itfBaseLoggerElementConnector <> 0 AND
	THIS^.itfBaseComponentConnector	<> 0 AND
	THIS^.itfBaseControlElementConnector <> 0 AND
	THIS^.itfBaseGroupElementConnector <> 0 AND
	THIS^.itfBaseTopElementConnector <> 0 AND
	THIS^.itfBaseLoggerConnector <> 0) THEN
	THIS^.bIsInit						:= TRUE;
END_IF
END_METHOD

METHOD LinkTopElementData : BOOL
VAR_INPUT
	stData				: REFERENCE TO ST_TopElement_HMI_Link;
END_VAR
THIS^.refstTopElementData	REF= stData.stTopElement;

THIS^.refstBaseLoggerElementDataHMI	REF= stData.stBaseLoggerElement;
THIS^.refstBaseComponentDataHMI		REF= stData.stBaseComponent;
THIS^.refstBaseControlElementDataHMI	REF= stData.stBaseControlElement;
THIS^.refstBaseGroupElementDataHMI		REF= stData.stBaseGroupElement;
THIS^.refstBaseTopElementDataHMI		REF= stData.stBaseTopElement;

THIS^.itfControlElement1.LinkControlElementData (stData := stData.stControlElement1);
THIS^.itfControlElement2.LinkControlElementData (stData := stData.stControlElement2);
THIS^.itfGroupElement1.LinkGroupelementData (stData := stData.stGroupElement1);
THIS^.itfComponent1.LinkComponentData (stData := stData.stComponent1);
THIS^.itfComponent2.LinkComponentData (stData := stData.stComponent2);
THIS^.itfComponent3.LinkComponentData (stData := stData.stComponent3);

THIS^.CreateLinkToEventsMemory ();



IF (__ISVALIDREF (THIS^.refstTopElementData) AND this^.IsLinkedReferences ()) THEN
	THIS^.bIsValidData		:= TRUE;
	LinkTopElementData		:= TRUE;
END_IF
END_METHOD

END_FUNCTION_BLOCK

// ---- POUs/A0_BaseFB/Command/FB_CommandTest.TcPOU
FUNCTION_BLOCK FB_CommandTest EXTENDS TcUnit.FB_TestSuite
VAR
	sText			: STRING;
	iCounter		: INT;
END_VAR


T01_TestPoleceniaProstego ();
T02_TestPoleceniaZlozonego ();

METHOD PUBLIC MetodaDlaPolecenbiaProstego : bool
VAR_INPUT
END_VAR
THIS^.sText := 'jestem w tej metodzie';
iCounter := iCounter + 1;
MetodaDlaPolecenbiaProstego	:= FALSE;
END_METHOD

METHOD PROTECTED T01_TestPoleceniaProstego
VAR_INPUT
END_VAR
IF (TcUnit.TEST_ORDERED ('T01_TestPoleceniaProstego')) THEN
	GVL.fbCommandEasy.Test ();
	AssertTrue (Condition := GVL.fbCommandEasy.IsStatus (), 	Message := 'T01a - Bledny status');
	AssertFalse (Condition := GVL.fbCommandEasy.IsBusy (),		Message := 'T01b - Bledny stan');
	GVL.fbCommandEasy.Execute ();
	GVL.fbCommandEasy.Test ();
	AssertFalse (Condition := GVL.fbCommandEasy.IsStatus (), 	Message := 'T02a - Bledny status');
	AssertTrue (Condition := GVL.fbCommandEasy.IsBusy (),		Message := 'T02b - Bledny stan');
	
	GVL.fbCommandEasy.OperationExecute ();
	GVL.fbCommandEasy.Operation (bIN := MetodaDlaPolecenbiaProstego ());
	
	AssertTrue (Condition := GVL.fbCommandEasy.IsFirstCycle (),Message := 'T03a - Bledny stan pierwszego przejscia');
	AssertTrue (Condition := GVL.fbCommandEasy.IsLastCycle (),	Message := 'T03b - Bledny stan ostatniego przejscia');
	
	GVL.fbCommandEasy.OperationExecute ();
	
	AssertFalse (Condition := GVL.fbCommandEasy.IsFirstCycle (),	Message := 'T04a - Bledny stan pierwszego przejscia');
	AssertFalse (Condition := GVL.fbCommandEasy.IsLastCycle (),		Message := 'T04b - Bledny stan ostatniego przejscia');

	GVL.fbCommandEasy.OperationExecute ();
	
	AssertFalse (Condition := GVL.fbCommandEasy.IsLastCycle (),	Message := 'T05a - Bledny stan pierwszego przejscia');
	AssertTrue (Condition := GVL.fbCommandEasy.IsStatus (),		Message := 'T05b - Bledny stan statusy');
	
	TcUnit.TEST_FINISHED ();
END_IF
END_METHOD

METHOD PROTECTED T02_TestPoleceniaZlozonego : BOOL

VAR
	bResult: BOOL;
END_VAR
IF (TcUnit.TEST_ORDERED ('T02_TestPolecenia')) THEN
	GVL.fbCommand.Test ();
	AssertTrue (Condition := GVL.fbCommand.IsStatus (), 	Message := 'T01a - Bledny status');
	AssertFalse (Condition := GVL.fbCommand.IsBusy (),		Message := 'T01b - Bledny stan');
	
	GVL.fbCommand.Execute ();
	GVL.fbCommand.Test ();
	AssertFalse (Condition := GVL.fbCommand.IsStatus (), 	Message := 'T02a - Bledny status');
	AssertTrue (Condition := GVL.fbCommand.IsBusy (),		Message := 'T02b - Bledny stan');
	
	IF (GVL.fbCommand.OperationExecute ()) THEN;
		bResult				:= TRUE;
		GVL.fbCommand.Operation (bIN := GVL.fbCommand.CyklTestu ());
	ELSE
		bResult				:= FALSE;
	END_IF
	AssertTrue (Condition := GVL.fbCommand.IsFirstCycle (),Message := 'T03a - Bledny stan pierwszego przejscia');
	AssertFalse (Condition := GVL.fbCommand.IsLastCycle (),Message := 'T03b - Bledny stan ostatniego przejscia');
	AssertFalse (Condition := bResult, 						Message := 'T03c - Bledny wynik');
	
	IF (GVL.fbCommand.OperationExecute ()) THEN;
		bResult				:= TRUE;
		GVL.fbCommand.Operation (bIN := GVL.fbCommand.CyklTestu ());
	ELSE
		bResult				:= FALSE;
	END_IF
	AssertFalse (Condition := GVL.fbCommand.IsFirstCycle (),	Message := 'T04a - Bledny stan pierwszego przejscia');
	AssertFalse (Condition := GVL.fbCommand.IsLastCycle (),	Message := 'T04b - Bledny stan ostatniego przejscia');
	AssertTrue (Condition := bResult, 							Message := 'T04c - Bledny wynik');
	
	WRITE_PROTECTED_BOOL (Ptr := ADR (GVL.fbCommand.bFinish), Value := TRUE);
	IF (GVL.fbCommand.OperationExecute ()) THEN;
		bResult				:= TRUE;
		GVL.fbCommand.Operation (bIN := GVL.fbCommand.CyklTestu ());
	ELSE
		bResult				:= FALSE;
	END_IF
	AssertFalse (Condition := GVL.fbCommand.IsFirstCycle (),	Message := 'T05a - Bledny stan pierwszego przejscia');
	Asserttrue (Condition := GVL.fbCommand.IsLastCycle (),		Message := 'T05b - Bledny stan ostatniego przejscia');
	AssertTrue (Condition := bResult, 							Message := 'T05c - Bledny wynik');
	
	IF (GVL.fbCommand.OperationExecute ()) THEN;
		bResult				:= TRUE;
		GVL.fbCommand.Operation (bIN := GVL.fbCommand.CyklTestu ());
	ELSE
		bResult				:= FALSE;
	END_IF
	AssertFalse (Condition := GVL.fbCommand.IsFirstCycle (),	Message := 'T06a - Bledny stan pierwszego przejscia');
	AssertFalse (Condition := GVL.fbCommand.IsLastCycle (),	Message := 'T06b - Bledny stan ostatniego przejscia');
	AssertFalse (Condition := bResult, 							Message := 'T06c - Bledny wynik');

	

	TcUnit.TEST_FINISHED ();
END_IF
END_METHOD

END_FUNCTION_BLOCK

// ---- POUs/A2_logger/FB_LoggerTest.TcPOU
FUNCTION_BLOCK FB_LoggerTest EXTENDS TcUnit.FB_TestSuite
VAR

END_VAR


T01_TestDodawaniaZgloszen ();
T02_TestDodawaniaZgloszen2 ();
T03_TestDodawaniaZgloszen3 ();
T04_TestDodawaniaKomponentowDoLogera ();

METHOD PRIVATE T01_TestDodawaniaZgloszen
VAR
	sttmpEvent: ST_BaseEvents_RowInQueue;
END_VAR
IF (TcUnit.TEST_ORDERED ('T01_TestDodawaniaZgloszen')) THEN
	WRITE_PROTECTED_BOOL (Ptr := ADR (GVL.fbLogger.bClearMemory), Value := TRUE);
	GVL.fbLogger ();
	AssertEquals_INT (Expected := 0, Actual := GVL.fbLogger.stBuffer.iNumerOfEvents, 	Message := 'T01a - bledna ilosc w kolejce');
	AssertEquals_INT (Expected := 0, Actual := GVL.fbLogger.stmemory.iNumberOfRow,		Message := 'T01b - bledna ilosc zgloszen');
//wyslanie zgloszenia 
	sttmpEvent.bActive				:= TRUE;
	sttmpEvent.bConfirm				:= TRUE;
	sttmpEvent.bIgnoreRepetitions	:= TRUE;
	sttmpEvent.dtStart				:= DT#2025-09-25-01:00:00;
	sttmpEvent.eEventCategory		:= E_BaseEvents_Category.Error;
	sttmpEvent.eEventAction			:= E_BaseEvents_Action.Start;
	sttmpEvent.uiIDEvent			:= 1;
	sttmpEvent.uiIDItem				:= 2;
	GVL.fbLogger.ReportEvent (stEvent := sttmpEvent);
	AssertEquals_INT (Expected := 1, Actual := GVL.fbLogger.stBuffer.iNumerOfEvents, 	Message := 'T02a - bledna ilosc w kolejce');
	AssertEquals_INT (Expected := 0, Actual := GVL.fbLogger.stmemory.iNumberOfRow,		Message := 'T02b - bledna ilosc zgloszen');
	GVL.fbLogger ();
	AssertEquals_INT (Expected := 0, Actual := GVL.fbLogger.stBuffer.iNumerOfEvents, 					Message := 'T03a - bledna ilosc w kolejce');
	AssertEquals_INT (Expected := 1, Actual := GVL.fbLogger.stmemory.iNumberOfRow,						Message := 'T03b - bledna ilosc zgloszen');
	AssertEquals_INT (Expected := 1, Actual := GVL.fbLogger.stNumberOfReports.iNumberOfActive,			Message := 'T03c - bledna ilosc zgloszen');
	AssertTrue (Condition := GVL.fbLogger.stNumberOfReports.arrActive [E_BaseEvents_Category.Error],	Message := 'T03d - bledny stan');
	AssertFalse (Condition := GVL.fbLogger.stNumberOfReports.arrActive [E_BaseEvents_Category.Alarm],	Message := 'T03d - bledny stan');
	AssertTrue (Condition := GVL.fbLogger.stNumberOfReports.bIsActive,									Message := 'T03e - bledny stan');
	AssertEquals_INT (Expected := 1, Actual := GVL.fbLogger.stNumberOfReports.iTotalNumer,				Message := 'T03f - bledna ilosc zgloszen');
//potwierdzenie zgloszenia 
	sttmpEvent.eEventAction			:= E_BaseEvents_Action.Confirm;
	sttmpEvent.uiIDEvent			:= 1;
	sttmpEvent.uiIDItem				:= 2;
	sttmpEvent.dtConfirmed			:= DT#2025-09-25-01:01:00;
	GVL.fbLogger.ReportEvent (stEvent := sttmpEvent);
	AssertEquals_INT (Expected := 1, Actual := GVL.fbLogger.stBuffer.iNumerOfEvents, 					Message := 'T04a - bledna ilosc w kolejce');
	AssertEquals_INT (Expected := 1, Actual := GVL.fbLogger.stmemory.iNumberOfRow,						Message := 'T04b - bledna ilosc zgloszen');
	GVL.fbLogger ();
	AssertEquals_INT (Expected := 0, Actual := GVL.fbLogger.stBuffer.iNumerOfEvents, 					Message := 'T05a - bledna ilosc w kolejce');
	AssertEquals_INT (Expected := 1, Actual := GVL.fbLogger.stmemory.iNumberOfRow,						Message := 'T05b - bledna ilosc zgloszen');
	AssertEquals_INT (Expected := 1, Actual := GVL.fbLogger.stNumberOfReports.iNumberOfActive,			Message := 'T05c - bledna ilosc zgloszen');
	AssertTrue (Condition := GVL.fbLogger.stNumberOfReports.arrActive [E_BaseEvents_Category.Error],	Message := 'T05d - bledny stan');
	AssertFalse (Condition := GVL.fbLogger.stNumberOfReports.arrActive [E_BaseEvents_Category.Alarm],	Message := 'T05d - bledny stan');
	AssertTrue (Condition := GVL.fbLogger.stNumberOfReports.bIsActive,									Message := 'T05e - bledny stan');
	AssertEquals_INT (Expected := 1, Actual := GVL.fbLogger.stNumberOfReports.iTotalNumer,				Message := 'T05f - bledna ilosc zgloszen');
//zamkniecie zgloszenia 
	sttmpEvent.eEventAction			:= E_BaseEvents_Action.Stop;
	sttmpEvent.uiIDEvent			:= 1;
	sttmpEvent.uiIDItem				:= 2;
	sttmpEvent.dtFinish				:= DT#2025-09-25-01:02:00;
	GVL.fbLogger.ReportEvent (stEvent := sttmpEvent);
	AssertEquals_INT (Expected := 1, Actual := GVL.fbLogger.stBuffer.iNumerOfEvents, 					Message := 'T04a - bledna ilosc w kolejce');
	AssertEquals_INT (Expected := 1, Actual := GVL.fbLogger.stmemory.iNumberOfRow,						Message := 'T04b - bledna ilosc zgloszen');
	GVL.fbLogger ();
	AssertEquals_INT (Expected := 0, Actual := GVL.fbLogger.stBuffer.iNumerOfEvents, 					Message := 'T05a - bledna ilosc w kolejce');
	AssertEquals_INT (Expected := 1, Actual := GVL.fbLogger.stmemory.iNumberOfRow,						Message := 'T05b - bledna ilosc zgloszen');
	AssertEquals_INT (Expected := 0, Actual := GVL.fbLogger.stNumberOfReports.iNumberOfActive,			Message := 'T05c - bledna ilosc zgloszen');
	AssertFalse (Condition := GVL.fbLogger.stNumberOfReports.arrActive [E_BaseEvents_Category.Error],	Message := 'T05d - bledny stan');
	AssertFalse (Condition := GVL.fbLogger.stNumberOfReports.arrActive [E_BaseEvents_Category.Alarm],	Message := 'T05d - bledny stan');
	Assertfalse (Condition := GVL.fbLogger.stNumberOfReports.bIsActive,									Message := 'T05e - bledny stan');
	AssertEquals_INT (Expected := 1, Actual := GVL.fbLogger.stNumberOfReports.iTotalNumer,				Message := 'T05f - bledna ilosc zgloszen');
	
	
	TcUnit.TEST_FINISHED ();
END_IF
END_METHOD

METHOD PRIVATE T02_TestDodawaniaZgloszen2
VAR
	sttmpEvent: ST_BaseEvents_RowInQueue;
END_VAR
IF (TcUnit.TEST_ORDERED ('T02_TestDodawaniaZgloszen2')) THEN
	GVL.fbLogger ();
	AssertEquals_INT (Expected := 0, Actual := GVL.fbLogger.stBuffer.iNumerOfEvents, 	Message := 'T01a - bledna ilosc w kolejce');
	AssertEquals_INT (Expected := 1, Actual := GVL.fbLogger.stmemory.iNumberOfRow,		Message := 'T01b - bledna ilosc zgloszen');
//wyslanie zgloszenia 
	sttmpEvent.bActive				:= TRUE;
	sttmpEvent.bConfirm				:= TRUE;
	sttmpEvent.bIgnoreRepetitions	:= TRUE;
	sttmpEvent.dtStart				:= DT#2025-09-25-02:00:00;
	sttmpEvent.eEventCategory		:= E_BaseEvents_Category.Error;
	sttmpEvent.eEventAction			:= E_BaseEvents_Action.Start;
	sttmpEvent.uiIDEvent			:= 1;
	sttmpEvent.uiIDItem				:= 2;
	GVL.fbLogger.ReportEvent (stEvent := sttmpEvent);
	AssertEquals_INT (Expected := 1, Actual := GVL.fbLogger.stBuffer.iNumerOfEvents, 					Message := 'T02a - bledna ilosc w kolejce');
	AssertEquals_INT (Expected := 1, Actual := GVL.fbLogger.stmemory.iNumberOfRow,						Message := 'T02b - bledna ilosc zgloszen');
	GVL.fbLogger ();
	AssertEquals_INT (Expected := 0, Actual := GVL.fbLogger.stBuffer.iNumerOfEvents, 					Message := 'T03a - bledna ilosc w kolejce');
	AssertEquals_INT (Expected := 2, Actual := GVL.fbLogger.stmemory.iNumberOfRow,						Message := 'T03b - bledna ilosc zgloszen');
	AssertEquals_INT (Expected := 1, Actual := GVL.fbLogger.stNumberOfReports.iNumberOfActive,			Message := 'T03c - bledna ilosc zgloszen');
	AssertTrue (Condition := GVL.fbLogger.stNumberOfReports.arrActive [E_BaseEvents_Category.Error],	Message := 'T03d - bledny stan');
	AssertFalse (Condition := GVL.fbLogger.stNumberOfReports.arrActive [E_BaseEvents_Category.Alarm],	Message := 'T03d - bledny stan');
	AssertTrue (Condition := GVL.fbLogger.stNumberOfReports.bIsActive,									Message := 'T03e - bledny stan');
	AssertEquals_INT (Expected := 2, Actual := GVL.fbLogger.stNumberOfReports.iTotalNumer,				Message := 'T03f - bledna ilosc zgloszen');
//zamkniecie zgloszenia  bez potwierdzenia a wymagane nic się nei powinno stać
	sttmpEvent.eEventAction			:= E_BaseEvents_Action.Stop;
	sttmpEvent.uiIDEvent			:= 1;
	sttmpEvent.uiIDItem				:= 2;
	sttmpEvent.dtFinish				:= DT#2025-09-25-02:00:00;
	GVL.fbLogger.ReportEvent (stEvent := sttmpEvent);
	AssertEquals_INT (Expected := 1, Actual := GVL.fbLogger.stBuffer.iNumerOfEvents, 					Message := 'T04a - bledna ilosc w kolejce');
	AssertEquals_INT (Expected := 2, Actual := GVL.fbLogger.stmemory.iNumberOfRow,						Message := 'T04b - bledna ilosc zgloszen');
	GVL.fbLogger ();
	AssertEquals_INT (Expected := 0, Actual := GVL.fbLogger.stBuffer.iNumerOfEvents, 					Message := 'T05a - bledna ilosc w kolejce');
	AssertEquals_INT (Expected := 2, Actual := GVL.fbLogger.stmemory.iNumberOfRow,						Message := 'T05b - bledna ilosc zgloszen');
	AssertEquals_INT (Expected := 1, Actual := GVL.fbLogger.stNumberOfReports.iNumberOfActive,			Message := 'T05c - bledna ilosc zgloszen');
	AssertTrue (Condition := GVL.fbLogger.stNumberOfReports.arrActive [E_BaseEvents_Category.Error],	Message := 'T05d - bledny stan');
	AssertFalse (Condition := GVL.fbLogger.stNumberOfReports.arrActive [E_BaseEvents_Category.Alarm],	Message := 'T05d - bledny stan');
	AssertTrue (Condition := GVL.fbLogger.stNumberOfReports.bIsActive,									Message := 'T05e - bledny stan');
	AssertEquals_INT (Expected := 2, Actual := GVL.fbLogger.stNumberOfReports.iTotalNumer,				Message := 'T05f - bledna ilosc zgloszen');
//potwierdzenie zgloszenia 
	sttmpEvent.eEventAction			:= E_BaseEvents_Action.Confirm;
	sttmpEvent.uiIDEvent			:= 1;
	sttmpEvent.uiIDItem				:= 2;
	sttmpEvent.dtConfirmed			:= DT#2025-09-25-02:01:00;
	GVL.fbLogger.ReportEvent (stEvent := sttmpEvent);
	AssertEquals_INT (Expected := 1, Actual := GVL.fbLogger.stBuffer.iNumerOfEvents, 					Message := 'T06a - bledna ilosc w kolejce');
	AssertEquals_INT (Expected := 2, Actual := GVL.fbLogger.stmemory.iNumberOfRow,						Message := 'T06b - bledna ilosc zgloszen');
	GVL.fbLogger ();
	AssertEquals_INT (Expected := 0, Actual := GVL.fbLogger.stBuffer.iNumerOfEvents, 					Message := 'T07a - bledna ilosc w kolejce');
	AssertEquals_INT (Expected := 2, Actual := GVL.fbLogger.stmemory.iNumberOfRow,						Message := 'T07b - bledna ilosc zgloszen');
	AssertEquals_INT (Expected := 1, Actual := GVL.fbLogger.stNumberOfReports.iNumberOfActive,			Message := 'T07c - bledna ilosc zgloszen');
	AssertTrue (Condition := GVL.fbLogger.stNumberOfReports.arrActive [E_BaseEvents_Category.Error],	Message := 'T07d - bledny stan');
	AssertFalse (Condition := GVL.fbLogger.stNumberOfReports.arrActive [E_BaseEvents_Category.Alarm],	Message := 'T07d - bledny stan');
	AssertTrue (Condition := GVL.fbLogger.stNumberOfReports.bIsActive,									Message := 'T07e - bledny stan');
	AssertEquals_INT (Expected := 2, Actual := GVL.fbLogger.stNumberOfReports.iTotalNumer,				Message := 'T07f - bledna ilosc zgloszen');
//zamkniecie zgloszenia 
	sttmpEvent.eEventAction			:= E_BaseEvents_Action.Stop;
	sttmpEvent.uiIDEvent			:= 1;
	sttmpEvent.uiIDItem				:= 2;
	sttmpEvent.dtFinish				:= DT#2025-09-25-02:02:00;
	GVL.fbLogger.ReportEvent (stEvent := sttmpEvent);
	AssertEquals_INT (Expected := 1, Actual := GVL.fbLogger.stBuffer.iNumerOfEvents, 					Message := 'T08a - bledna ilosc w kolejce');
	AssertEquals_INT (Expected := 2, Actual := GVL.fbLogger.stmemory.iNumberOfRow,						Message := 'T08b - bledna ilosc zgloszen');
	GVL.fbLogger ();
	AssertEquals_INT (Expected := 0, Actual := GVL.fbLogger.stBuffer.iNumerOfEvents, 					Message := 'T09a - bledna ilosc w kolejce');
	AssertEquals_INT (Expected := 2, Actual := GVL.fbLogger.stmemory.iNumberOfRow,						Message := 'T09b - bledna ilosc zgloszen');
	AssertEquals_INT (Expected := 0, Actual := GVL.fbLogger.stNumberOfReports.iNumberOfActive,			Message := 'T09c - bledna ilosc zgloszen');
	AssertFalse (Condition := GVL.fbLogger.stNumberOfReports.arrActive [E_BaseEvents_Category.Error],	Message := 'T09d - bledny stan');
	AssertFalse (Condition := GVL.fbLogger.stNumberOfReports.arrActive [E_BaseEvents_Category.Alarm],	Message := 'T09d - bledny stan');
	Assertfalse (Condition := GVL.fbLogger.stNumberOfReports.bIsActive,									Message := 'T09e - bledny stan');
	AssertEquals_INT (Expected := 2, Actual := GVL.fbLogger.stNumberOfReports.iTotalNumer,				Message := 'T09f - bledna ilosc zgloszen');
	
	
	TcUnit.TEST_FINISHED ();
END_IF
END_METHOD

METHOD PRIVATE T03_TestDodawaniaZgloszen3
VAR
	sttmpEvent: ST_BaseEvents_RowInQueue;
END_VAR
IF (TcUnit.TEST_ORDERED ('T03_TestDodawaniaZgloszen3')) THEN
//wyslanie zgloszenia 
	sttmpEvent.bActive				:= TRUE;
	sttmpEvent.bConfirm				:= FALSE;
	sttmpEvent.bIgnoreRepetitions	:= FALSE;
	sttmpEvent.dtStart				:= DT#2025-09-25-03:00:00;
	sttmpEvent.eEventCategory		:= E_BaseEvents_Category.Alarm;
	sttmpEvent.eEventAction			:= E_BaseEvents_Action.Start;
	sttmpEvent.uiIDEvent			:= 1;
	sttmpEvent.uiIDItem				:= 1;
	GVL.fbLogger.ReportEvent (stEvent := sttmpEvent);
	GVL.fbLogger ();
//zamkniecie zgloszenia 
	sttmpEvent.eEventAction			:= E_BaseEvents_Action.Stop;
	sttmpEvent.uiIDEvent			:= 1;
	sttmpEvent.uiIDItem				:= 1;
	sttmpEvent.dtFinish				:= DT#2025-09-25-03:02:00;
	GVL.fbLogger.ReportEvent (stEvent := sttmpEvent);
	GVL.fbLogger ();
//wyslanie zgloszenia 
	sttmpEvent.bActive				:= TRUE;
	sttmpEvent.bConfirm				:= FALSE;
	sttmpEvent.bIgnoreRepetitions	:= FALSE;
	sttmpEvent.dtStart				:= DT#2025-09-25-03:10:00;
	sttmpEvent.eEventCategory		:= E_BaseEvents_Category.Alarm;
	sttmpEvent.eEventAction			:= E_BaseEvents_Action.Start;
	sttmpEvent.uiIDEvent			:= 1;
	sttmpEvent.uiIDItem				:= 1;
	GVL.fbLogger.ReportEvent (stEvent := sttmpEvent);
	GVL.fbLogger ();
//wyslanie zgloszenia 
	sttmpEvent.bActive				:= TRUE;
	sttmpEvent.bConfirm				:= TRUE;
	sttmpEvent.bIgnoreRepetitions	:= TRUE;
	sttmpEvent.dtStart				:= DT#2025-09-25-03:20:00;
	sttmpEvent.eEventCategory		:= E_BaseEvents_Category.Error;
	sttmpEvent.eEventAction			:= E_BaseEvents_Action.Start;
	sttmpEvent.uiIDEvent			:= 2;
	sttmpEvent.uiIDItem				:= 1;
	GVL.fbLogger.ReportEvent (stEvent := sttmpEvent);
	GVL.fbLogger ();
//potwierdzenie zgloszenia 
	sttmpEvent.eEventAction			:= E_BaseEvents_Action.Confirm;
	sttmpEvent.uiIDEvent			:= 2;
	sttmpEvent.uiIDItem				:= 1;
	sttmpEvent.dtConfirmed			:= DT#2025-09-25-03:21:00;
	GVL.fbLogger.ReportEvent (stEvent := sttmpEvent);
	GVL.fbLogger ();
//zamkniecie zgloszenia 
	sttmpEvent.eEventAction			:= E_BaseEvents_Action.Stop;
	sttmpEvent.uiIDEvent			:= 2;
	sttmpEvent.uiIDItem				:= 1;
	sttmpEvent.dtFinish				:= DT#2025-09-25-03:22:00;
	GVL.fbLogger.ReportEvent (stEvent := sttmpEvent);
	GVL.fbLogger ();
//wyslanie zgloszenia 
	sttmpEvent.bActive				:= TRUE;
	sttmpEvent.bConfirm				:= FALSE;
	sttmpEvent.bIgnoreRepetitions	:= TRUE;
	sttmpEvent.dtStart				:= DT#2025-09-25-04:00:00;
	sttmpEvent.eEventCategory		:= E_BaseEvents_Category.Error;
	sttmpEvent.eEventAction			:= E_BaseEvents_Action.Start;
	sttmpEvent.uiIDEvent			:= 3;
	sttmpEvent.uiIDItem				:= 1;
	GVL.fbLogger.ReportEvent (stEvent := sttmpEvent);
	GVL.fbLogger ();
//wyslanie zgloszenia 
	sttmpEvent.bActive				:= TRUE;
	sttmpEvent.bConfirm				:= FALSE;
	sttmpEvent.bIgnoreRepetitions	:= TRUE;
	sttmpEvent.dtStart				:= DT#2025-09-25-04:20:00;
	sttmpEvent.eEventCategory		:= E_BaseEvents_Category.Message;
	sttmpEvent.eEventAction			:= E_BaseEvents_Action.Start;
	sttmpEvent.uiIDEvent			:= 4;
	sttmpEvent.uiIDItem				:= 1;
	GVL.fbLogger.ReportEvent (stEvent := sttmpEvent);
	GVL.fbLogger ();
//zamkniecie zgloszenia 
	sttmpEvent.eEventAction			:= E_BaseEvents_Action.Stop;
	sttmpEvent.uiIDEvent			:= 4;
	sttmpEvent.uiIDItem				:= 1;
	sttmpEvent.dtFinish				:= DT#2025-09-25-04:22:00;
	GVL.fbLogger.ReportEvent (stEvent := sttmpEvent);
	GVL.fbLogger ();
	
	
	TcUnit.TEST_FINISHED ();
END_IF
END_METHOD

METHOD PROTECTED T04_TestDodawaniaKomponentowDoLogera
VAR_INPUT
END_VAR
IF (TcUnit.TEST_ORDERED ('T04_TestDodawaniaKomponentowDoLogera')) THEN
	GVL_Variable.fbComponent_1_L.SetID (uiID 	:= 1);
	GVL_Variable.fbComponent_2_L.SetID (uiID 	:= 2);
	GVL_Variable.fbComponent_3_L.SetID (uiID 	:= 3);
	

	GVL.fbLogger.AddItem (itfItem := GVL_Variable.fbComponent_1_L);
	GVL.fbLogger.AddItem (itfItem := GVL_Variable.fbComponent_2_L);
	GVL.fbLogger.AddItem (itfItem := GVL_Variable.fbComponent_3_L);
	
//dodać testowanie dodawania FB_Control FB_Group i FB_Top	
	TcUnit.TEST_FINISHED ();
END_IF
END_METHOD

END_FUNCTION_BLOCK

// ---- POUs/A8_CommunicatorTest/FB_CommunicatorClient.TcPOU
FUNCTION_BLOCK FB_CommunicatorClient EXTENDS FB_BaseGroupElement
VAR
END_VAR

METHOD PUBLIC Confirm : BOOL
VAR_INPUT
	sText: STRING;
END_VAR
Confirm		:= THIS^.itfCommunicator.ReceiveDataConfirm (sText := sText, itfRecipient := this^);
END_METHOD

METHOD PUBLIC ReceiveMessage : BOOL
VAR_INPUT
	sText: STRING;
END_VAR

VAR_OUTPUT
	bValue: BOOL;
END_VAR
ReceiveMessage		:= THIS^.itfCommunicator.ReceiveData_BOOL (sText := sText, itfRecipient := THIS^, bValue => bValue);
END_METHOD

METHOD PUBLIC SendMessage : BOOL
VAR_INPUT
	sText: STRING;
END_VAR
SendMessage	:= THIS^.itfCommunicator.SendData_BOOL (sText := sText, itfSender := THIS^);
END_METHOD

END_FUNCTION_BLOCK

// ---- POUs/FB_ItemTest.TcPOU
FUNCTION_BLOCK FB_ItemTest EXTENDS TcUnit.FB_TestSuite
VAR
END_VAR

T01_TestAddItems ();
T02_TestFirstCycle ();
T03_TestSetidEvent ();
T04_TestSetIditem ();
T05_TestSetCodeItem ();
T06_TestEventsAdd ();
T07_TestLinkData ();
T08_TestEventReport ();
T09_TestEventReport ();
T10_PreparetableEventsForTesting ();

T11_TestGenerateListEvent ();

T12_TestPower ();
T13_TestPowerForTopElement ();

//T14_TestHomingControlElementWithouutHomingMethod ();
//T15_TestHomingControlElementWithHomingMetod ();
//T16_TestingTopElementHoming ();

T20_TestCommunicator ();
T21_TestCreateTepmplate ();
T22_TestAddRecipeFromTemplate ();
T23_TestDeleteRecipe ();
T24_TestCopyRecipeToNewRecipe ();

//T99_Test ();

METHOD PRIVATE T01_TestAddItems
VAR_INPUT
END_VAR
IF (TcUnit.TEST_ORDERED ('T01_TestAddItems')) THEN
	AssertEquals_UINT (Expected := 3, Actual := GVL_Variable.fbPB1.uiNumberOfComponents, 		Message := 'T01 - bledna ilosc elementow');
	AssertEquals_UINT (Expected := 3, Actual := GVL_Variable.fbPB1.uiNumberOfControlElement, 	Message := 'T02 - bledna ilosc elementow');

	AssertEquals_UINT (Expected := 2, Actual := GVL_Variable.fbPB1_ZL1.uiNumberOfComponents, 	Message := 'T03 - bledna ilosc elementow');
	AssertEquals_UINT (Expected := 2, Actual := GVL_Variable.fbPB1_ZL1.uiNumberOfControlElement,Message := 'T04 - bledna ilosc elementow');
	
	AssertEquals_UINT (Expected := 2, Actual := GVL_Variable.fbPB1_Wyk1.uiNumberOfComponents, 	Message := 'T05 - bledna ilosc elementow');
	AssertEquals_UINT (Expected := 2, Actual := GVL_Variable.fbPB1_Wyk2.uiNumberOfComponents, 	Message := 'T06 - bledna ilosc elementow');
	

	TcUnit.TEST_FINISHED ();
END_IF
END_METHOD

METHOD PRIVATE T02_TestFirstCycle
VAR_INPUT
END_VAR

VAR
	bResult: BOOL;
END_VAR
IF (TcUnit.TEST_ORDERED ('T02_TestFirstCycle')) THEN
	GVL.stCommonData.itfTime				:= GVL.fbMyTime;
	GVL.stCommonData.itfLocaciotn			:= GVL.fbMyLocation;
	GVL.stCommonData.itfLogger				:= GVL.fbLogger;
	
	bResult 	:= GVL_Variable.fbPB1.LinkCommonData (stCommonData	:= GVL.stCommonData);
	
	AssertTrue (Condition := bResult, Message := 'T01a - bladny wynik przepisania');
	
	bResult 	:= GVL_Variable.fbPB1.FirstCycle ();
	AssertTrue (Condition := bResult, Message := 'T02a - bladny wynik pierwszego przejścia');
	
	bResult		:= GVL_Variable.fbPB1.LinkSS1 (fbSS1		:= GVL.fbSS1);
	AssertTrue (Condition := bResult, Message := 'T03a - bladny wynik linkowania');
	
	bResult		:= GVL_Variable.fbPB1.LinkSTO (fbSTO		:= GVL.fbSTO);
	AssertTrue (Condition := bResult, Message := 'T03b - bladny wynik linkowania');
	
	
	
	TcUnit.TEST_FINISHED ();
END_IF
END_METHOD

METHOD PRIVATE T03_TestSetidEvent
VAR_INPUT
END_VAR

VAR
	uiLastID: UINT;
END_VAR
IF (TcUnit.TEST_ORDERED ('T03_TestSetidEvent')) THEN
	uiLastID		:= GVL_Variable.fbPB1.SetEventsIDs (uiNewID	:= 1);
	
	AssertEquals_UINT (Expected := 109, Actual := uiLastID, Message := 'T01 - Bledna ilosc nadanych ID zgloszeniom');
	//58 przekazywany do następnego defacto jest zgłoszęń o jeden mniej
	
	
	TcUnit.TEST_FINISHED ();
END_IF
END_METHOD

METHOD PRIVATE T04_TestSetIditem
VAR_INPUT
END_VAR

VAR
	uiResult: UINT;
END_VAR
IF (TcUnit.TEST_ORDERED ('T04_TestSetIditem')) THEN
	uiResult 	:= GVL_Variable.fbPB1.SetID (uiID := 1);
	AssertEquals_UINT (Expected := 19, Actual := uiResult, Message := 'T01 - bledny numer id');
	
	
	TcUnit.TEST_FINISHED ();
END_IF
END_METHOD

METHOD PRIVATE T05_TestSetCodeItem
VAR_INPUT
END_VAR

VAR
	sResult: string;
END_VAR
IF (TcUnit.TEST_ORDERED ('T05_TestSetCodeItem')) THEN
	GVL_Variable.fbPB1.SetCode (sCode := '0.0.0.0.0', sAdd := '1');
//	AssertEquals_UINT (Expected := 19, Actual := uiResult, Message := 'T01 - bledny numer id');
	AssertEquals_STRING (Expected := '1.0.0.0.0', Actual := GVL_Variable.fbPB1.GetCode (), Message := 'T01 - Bledny kod PB');

	AssertEquals_STRING (Expected := '1.1.0.0.0', Actual := GVL_Variable.fbPB1_K1.GetCode (), Message := 'T01 - Bledny kod PB K1');
	AssertEquals_STRING (Expected := '1.2.0.0.0', Actual := GVL_Variable.fbPB1_K2.GetCode (), Message := 'T02 - Bledny kod PB K2');
	AssertEquals_STRING (Expected := '1.3.0.0.0', Actual := GVL_Variable.fbPB1_K3.GetCode (), Message := 'T03 - Bledny kod PB K3');
	
	AssertEquals_STRING (Expected := '1.4.0.0.0', Actual := GVL_Variable.fbPB1_Wyk1.GetCode (), 	Message := 'T04 - Bledny kod PB WYK1');
	AssertEquals_STRING (Expected := '1.4.1.0.0', Actual := GVL_Variable.fbPB1_Wyk1_K1.GetCode (), 	Message := 'T05 - Bledny kod PB WYK1 K1');
	AssertEquals_STRING (Expected := '1.4.2.0.0', Actual := GVL_Variable.fbPB1_Wyk1_K2.GetCode (), 	Message := 'T06 - Bledny kod PB WYK1 K2');
	
	AssertEquals_STRING (Expected := '1.5.0.0.0', Actual := GVL_Variable.fbPB1_Wyk2.GetCode (), 	Message := 'T07 - Bledny kod PB WYK1');
	AssertEquals_STRING (Expected := '1.5.1.0.0', Actual := GVL_Variable.fbPB1_Wyk2_K1.GetCode (), 	Message := 'T08 - Bledny kod PB WYK1 K1');
	AssertEquals_STRING (Expected := '1.5.2.0.0', Actual := GVL_Variable.fbPB1_Wyk2_K2.GetCode (), 	Message := 'T09 - Bledny kod PB WYK1 K2');
	
	AssertEquals_STRING (Expected := '1.6.0.0.0', Actual := GVL_Variable.fbPB1_ZL1.GetCode (), 		Message := 'T10 - Bledny kod PB ZL1');
	AssertEquals_STRING (Expected := '1.6.1.0.0', Actual := GVL_Variable.fbPB1_ZL1_K1.GetCode (), 	Message := 'T11 - Bledny kod PB ZL1 K1');
	AssertEquals_STRING (Expected := '1.6.2.0.0', Actual := GVL_Variable.fbPB1_ZL1_K2.GetCode (), 	Message := 'T12 - Bledny kod PB ZL1 K2');
	
	AssertEquals_STRING (Expected := '1.6.3.0.0', Actual := GVL_Variable.fbPB1_ZL1_Wyk1.GetCode (), 	Message := 'T13 - Bledny kod PB ZL1 WYK1');
	AssertEquals_STRING (Expected := '1.6.3.1.0', Actual := GVL_Variable.fbPB1_ZL1_Wyk1_K1.GetCode (), 	Message := 'T14 - Bledny kod PB ZL1 WYK1 K1');
	AssertEquals_STRING (Expected := '1.6.3.2.0', Actual := GVL_Variable.fbPB1_ZL1_Wyk1_K2.GetCode (), 	Message := 'T15 - Bledny kod PB ZL1 WYK1 K2');
	
	AssertEquals_STRING (Expected := '1.6.4.0.0', Actual := GVL_Variable.fbPB1_ZL1_Wyk2.GetCode (), 	Message := 'T16 - Bledny kod PB ZL2 WYK1');
	AssertEquals_STRING (Expected := '1.6.4.1.0', Actual := GVL_Variable.fbPB1_ZL1_Wyk2_K1.GetCode (), 	Message := 'T17 - Bledny kod PB ZL2 WYK1 K1');
	AssertEquals_STRING (Expected := '1.6.4.2.0', Actual := GVL_Variable.fbPB1_ZL1_Wyk2_K2.GetCode (), 	Message := 'T18 - Bledny kod PB ZL2 WYK1 K2');
	
	TcUnit.TEST_FINISHED ();
END_IF
END_METHOD

METHOD PRIVATE T06_TestEventsAdd
VAR_INPUT
END_VAR
IF (TcUnit.TEST_ORDERED ('T06_TestEventsAdd')) THEN
	AssertEquals_UINT (Expected := 5, Actual := GVL_Variable.fbPB1.stEvents.uiNumberOfAdded, 	Message := 'T01 - bledna ilosc');
	
	AssertEquals_UINT (Expected := 6, Actual := GVL_Variable.fbPB1_K1.stEvents.uiNumberOfAdded, Message := 'T02 - bledna ilosc');
	AssertEquals_UINT (Expected := 6, Actual := GVL_Variable.fbPB1_K2.stEvents.uiNumberOfAdded, Message := 'T03 - bledna ilosc');
	AssertEquals_UINT (Expected := 6, Actual := GVL_Variable.fbPB1_K3.stEvents.uiNumberOfAdded, Message := 'T04 - bledna ilosc');
 	
	AssertEquals_UINT (Expected := 5, Actual := GVL_Variable.fbPB1_Wyk1.stEvents.uiNumberOfAdded, Message := 'T05 - bledna ilosc');
	AssertEquals_UINT (Expected := 5, Actual := GVL_Variable.fbPB1_Wyk2.stEvents.uiNumberOfAdded, Message := 'T06 - bledna ilosc');
	
	AssertEquals_UINT (Expected := 5, Actual := GVL_Variable.fbPB1_ZL1.stEvents.uiNumberOfAdded, Message := 'T07 - bledna ilosc');
	
	TcUnit.TEST_FINISHED ();
END_IF
END_METHOD

METHOD PRIVATE T07_TestLinkData
VAR_INPUT
END_VAR

VAR
	bResult: BOOL;
END_VAR
IF (TcUnit.TEST_ORDERED ('T07_TestLinkData')) THEN
	bResult 	:= GVL_VariableHMI.fbPB1_HMI.LinkCommonData (stCommonData	:= GVL.stCommonData);
	AssertTrue (Condition := bResult, Message := 'T01a - bladny wynik przepisania');
	
	GVL_VariableHMI.fbPB1_HMI.LinkTopElementData (stData := gvl.stTopElementData);
	
	AssertTrue (Condition := GVL_VariableHMI.fbPB1_HMI.IsValidCommonData (), Message := 'T02 - bledna flaga podlaczenia danych wspólnych');
	
	bResult		:= GVL_Variable.fbPB1.JoinTheLogger ();
	AssertTrue (Condition := bResult, Message := 'T03 - bladny wynik przepisania');
	
	TcUnit.TEST_FINISHED ();
END_IF
END_METHOD

METHOD PRIVATE T08_TestEventReport
VAR_INPUT
END_VAR
IF (TcUnit.TEST_ORDERED ('T08_TestEventReport')) THEN
(*	Wyczyszenie pamięci i sprawdzenie czy rzeczywiście nic tam nie ma *)
	WRITE_PROTECTED_BOOL (Ptr := ADR (GVL.fbLogger.bClearMemory), Value := TRUE);
	GVL.fbLogger ();
	AssertEquals_INT (Expected := 0, Actual := GVL.fbLogger.stBuffer.iNumerOfEvents, 	Message := 'T01a - bledna ilosc w kolejce');
	AssertEquals_INT (Expected := 0, Actual := GVL.fbLogger.stmemory.iNumberOfRow,		Message := 'T01b - bledna ilosc zgloszen');
(*	Wyslanie zgloszen	*)
	WRITE_PROTECTED_BOOL (Ptr := ADR (GVL_Variable.fbPB1_K1.bSetAlarm), Value := TRUE);
	GVL_Variable.fbPB1_K1 ();
	AssertEquals_INT (Expected := 1, Actual := GVL.fbLogger.stBuffer.iNumerOfEvents, 					Message := 'T02a - bledna ilosc w kolejce');
	AssertEquals_INT (Expected := 0, Actual := GVL.fbLogger.stmemory.iNumberOfRow,						Message := 'T02b - bledna ilosc zgloszen');
	GVL.fbLogger ();
	AssertEquals_INT (Expected := 0, Actual := GVL.fbLogger.stBuffer.iNumerOfEvents, 					Message := 'T03a - bledna ilosc w kolejce');
	AssertEquals_INT (Expected := 1, Actual := GVL.fbLogger.stmemory.iNumberOfRow,						Message := 'T03b - bledna ilosc zgloszen');
	AssertEquals_INT (Expected := 1, Actual := GVL.fbLogger.stNumberOfReports.iNumberOfActive,			Message := 'T03c - bledna ilosc zgloszen');
	AssertFalse (Condition := GVL.fbLogger.stNumberOfReports.arrActive [E_BaseEvents_Category.Error],	Message := 'T03d - bledny stan');
	AssertTrue (Condition := GVL.fbLogger.stNumberOfReports.arrActive [E_BaseEvents_Category.Alarm],	Message := 'T03e - bledny stan');
	AssertTrue (Condition := GVL.fbLogger.stNumberOfReports.bIsActive,									Message := 'T03f - bledny stan');
	AssertEquals_INT (Expected := 1, Actual := GVL.fbLogger.stNumberOfReports.iTotalNumer,				Message := 'T03g - bledna ilosc zgloszen');
	AssertEquals_UINT (Expected := 2, Actual := GVL.fbLogger.stMemory.arrRow [1].uiIDItem,				Message := 'T03h - bledne ID elementu');
	AssertEquals_UINT (Expected := 7, Actual := GVL.fbLogger.stMemory.arrRow [1].uiIDEvent,				Message := 'T03i - bledne ID zgloszenia');
(*	Wyslanie zgloszen zamnięcie *)
	WRITE_PROTECTED_BOOL (Ptr := ADR (GVL_Variable.fbPB1_K1.bResetAlarm), Value := TRUE);
	GVL_Variable.fbPB1_K1 ();
	AssertEquals_INT (Expected := 1, Actual := GVL.fbLogger.stBuffer.iNumerOfEvents, 					Message := 'T04a - bledna ilosc w kolejce');
	AssertEquals_INT (Expected := 1, Actual := GVL.fbLogger.stmemory.iNumberOfRow,						Message := 'T04b - bledna ilosc zgloszen');
	GVL.fbLogger ();
	AssertEquals_INT (Expected := 0, Actual := GVL.fbLogger.stBuffer.iNumerOfEvents, 					Message := 'T05a - bledna ilosc w kolejce');
	AssertEquals_INT (Expected := 1, Actual := GVL.fbLogger.stmemory.iNumberOfRow,						Message := 'T05b - bledna ilosc zgloszen');
	AssertEquals_INT (Expected := 0, Actual := GVL.fbLogger.stNumberOfReports.iNumberOfActive,			Message := 'T05c - bledna ilosc zgloszen');
	AssertFalse (Condition := GVL.fbLogger.stNumberOfReports.arrActive [E_BaseEvents_Category.Error],	Message := 'T05d - bledny stan');
	AssertFalse (Condition := GVL.fbLogger.stNumberOfReports.arrActive [E_BaseEvents_Category.Alarm],	Message := 'T05e - bledny stan');
	AssertFalse (Condition := GVL.fbLogger.stNumberOfReports.bIsActive,									Message := 'T05f - bledny stan');
	AssertEquals_INT (Expected := 1, Actual := GVL.fbLogger.stNumberOfReports.iTotalNumer,				Message := 'T05g - bledna ilosc zgloszen');
	AssertEquals_UINT (Expected := 2, Actual := GVL.fbLogger.stMemory.arrRow [1].uiIDItem,				Message := 'T05h - bledne ID elementu');
	AssertEquals_UINT (Expected := 7, Actual := GVL.fbLogger.stMemory.arrRow [1].uiIDEvent,				Message := 'T05i - bledne ID zgloszenia');
(*	Wyslanie zgloszen	*)
	WRITE_PROTECTED_BOOL (Ptr := ADR (GVL_Variable.fbPB1_K1.bSetAlarm), Value := TRUE);
	GVL_Variable.fbPB1_K1 ();
	AssertEquals_INT (Expected := 1, Actual := GVL.fbLogger.stBuffer.iNumerOfEvents, 					Message := 'T06a - bledna ilosc w kolejce');
	AssertEquals_INT (Expected := 1, Actual := GVL.fbLogger.stmemory.iNumberOfRow,						Message := 'T06b - bledna ilosc zgloszen');
	GVL.fbLogger ();
	AssertEquals_INT (Expected := 0, Actual := GVL.fbLogger.stBuffer.iNumerOfEvents, 					Message := 'T07a - bledna ilosc w kolejce');
	AssertEquals_INT (Expected := 2, Actual := GVL.fbLogger.stmemory.iNumberOfRow,						Message := 'T07b - bledna ilosc zgloszen');
	AssertEquals_INT (Expected := 1, Actual := GVL.fbLogger.stNumberOfReports.iNumberOfActive,			Message := 'T07c - bledna ilosc zgloszen');
	AssertFalse (Condition := GVL.fbLogger.stNumberOfReports.arrActive [E_BaseEvents_Category.Error],	Message := 'T07d - bledny stan');
	AssertTrue (Condition := GVL.fbLogger.stNumberOfReports.arrActive [E_BaseEvents_Category.Alarm],	Message := 'T07e - bledny stan');
	AssertTrue (Condition := GVL.fbLogger.stNumberOfReports.bIsActive,									Message := 'T07f - bledny stan');
	AssertEquals_INT (Expected := 2, Actual := GVL.fbLogger.stNumberOfReports.iTotalNumer,				Message := 'T07g - bledna ilosc zgloszen');
	AssertEquals_UINT (Expected := 2, Actual := GVL.fbLogger.stMemory.arrRow [1].uiIDItem,				Message := 'T07h - 1 - bledne ID elementu');
	AssertEquals_UINT (Expected := 7, Actual := GVL.fbLogger.stMemory.arrRow [1].uiIDEvent,				Message := 'T07i - 2 - bledne ID zgloszenia');
	AssertEquals_UINT (Expected := 2, Actual := GVL.fbLogger.stMemory.arrRow [2].uiIDItem,				Message := 'T07j - 3 - bledne ID elementu');
	AssertEquals_UINT (Expected := 7, Actual := GVL.fbLogger.stMemory.arrRow [2].uiIDEvent,				Message := 'T07k - 4 - bledne ID zgloszenia');
(*	proba wysłania potwierrdzenia do zdarzenia bez potwierdzenia nic sie nie powinno wyfarzyć 	*)
	WRITE_PROTECTED_BOOL (Ptr := ADR (GVL_Variable.fbPB1_K1.bAckAlarm), Value := TRUE);
	GVL_Variable.fbPB1_K1 ();
	AssertEquals_INT (Expected := 1, Actual := GVL.fbLogger.stBuffer.iNumerOfEvents, 					Message := 'T08a - bledna ilosc w kolejce');
	AssertEquals_INT (Expected := 2, Actual := GVL.fbLogger.stmemory.iNumberOfRow,						Message := 'T08b - bledna ilosc zgloszen');
	GVL.fbLogger ();
	AssertEquals_INT (Expected := 0, Actual := GVL.fbLogger.stBuffer.iNumerOfEvents, 					Message := 'T09a - bledna ilosc w kolejce');
	AssertEquals_INT (Expected := 2, Actual := GVL.fbLogger.stmemory.iNumberOfRow,						Message := 'T09b - bledna ilosc zgloszen');
	AssertEquals_INT (Expected := 1, Actual := GVL.fbLogger.stNumberOfReports.iNumberOfActive,			Message := 'T09c - bledna ilosc zgloszen');
	AssertFalse (Condition := GVL.fbLogger.stNumberOfReports.arrActive [E_BaseEvents_Category.Error],	Message := 'T09d - bledny stan');
	AssertTrue (Condition := GVL.fbLogger.stNumberOfReports.arrActive [E_BaseEvents_Category.Alarm],	Message := 'T09e - bledny stan');
	AssertTrue (Condition := GVL.fbLogger.stNumberOfReports.bIsActive,									Message := 'T09f - bledny stan');
	AssertEquals_INT (Expected := 2, Actual := GVL.fbLogger.stNumberOfReports.iTotalNumer,				Message := 'T09g - bledna ilosc zgloszen');
	AssertEquals_UINT (Expected := 2, Actual := GVL.fbLogger.stMemory.arrRow [1].uiIDItem,				Message := 'T09h - 1 - bledne ID elementu');
	AssertEquals_UINT (Expected := 7, Actual := GVL.fbLogger.stMemory.arrRow [1].uiIDEvent,				Message := 'T09i - 2 - bledne ID zgloszenia');
	AssertEquals_UINT (Expected := 2, Actual := GVL.fbLogger.stMemory.arrRow [2].uiIDItem,				Message := 'T09j - 3 - bledne ID elementu');
	AssertEquals_UINT (Expected := 7, Actual := GVL.fbLogger.stMemory.arrRow [2].uiIDEvent,				Message := 'T09k - 4 - bledne ID zgloszenia');
	AssertFalse (Condition := gvl.fbLogger.stMemory.arrRow [1].bConfirm,								Message := 'T09l - bledny stan');
	AssertFalse (Condition := gvl.fbLogger.stMemory.arrRow [1].bConfirmed,								Message := 'T09m - bledny stan');
(*	Wyslanie zgloszen zamnięcie *)
	WRITE_PROTECTED_BOOL (Ptr := ADR (GVL_Variable.fbPB1_K1.bResetAlarm), Value := TRUE);
	GVL_Variable.fbPB1_K1 ();
	AssertEquals_INT (Expected := 1, Actual := GVL.fbLogger.stBuffer.iNumerOfEvents, 					Message := 'T10a - bledna ilosc w kolejce');
	AssertEquals_INT (Expected := 2, Actual := GVL.fbLogger.stmemory.iNumberOfRow,						Message := 'T10b - bledna ilosc zgloszen');
	GVL.fbLogger ();
	AssertEquals_INT (Expected := 0, Actual := GVL.fbLogger.stBuffer.iNumerOfEvents, 					Message := 'T11a - bledna ilosc w kolejce');
	AssertEquals_INT (Expected := 2, Actual := GVL.fbLogger.stmemory.iNumberOfRow,						Message := 'T11b - bledna ilosc zgloszen');
	AssertEquals_INT (Expected := 0, Actual := GVL.fbLogger.stNumberOfReports.iNumberOfActive,			Message := 'T11c - bledna ilosc zgloszen');
	AssertFalse (Condition := GVL.fbLogger.stNumberOfReports.arrActive [E_BaseEvents_Category.Error],	Message := 'T11d - bledny stan');
	AssertFalse (Condition := GVL.fbLogger.stNumberOfReports.arrActive [E_BaseEvents_Category.Alarm],	Message := 'T11e - bledny stan');
	AssertFalse (Condition := GVL.fbLogger.stNumberOfReports.bIsActive,									Message := 'T11f - bledny stan');
	AssertEquals_INT (Expected := 2, Actual := GVL.fbLogger.stNumberOfReports.iTotalNumer,				Message := 'T11g - bledna ilosc zgloszen');
	AssertEquals_UINT (Expected := 2, Actual := GVL.fbLogger.stMemory.arrRow [1].uiIDItem,				Message := 'T11h - 1 - bledne ID elementu');
	AssertEquals_UINT (Expected := 7, Actual := GVL.fbLogger.stMemory.arrRow [1].uiIDEvent,				Message := 'T11i - 2 - bledne ID zgloszenia');
	AssertEquals_UINT (Expected := 2, Actual := GVL.fbLogger.stMemory.arrRow [2].uiIDItem,				Message := 'T11j - 3 - bledne ID elementu');
	AssertEquals_UINT (Expected := 7, Actual := GVL.fbLogger.stMemory.arrRow [2].uiIDEvent,				Message := 'T11k - 4 - bledne ID zgloszenia');
	
	TcUnit.TEST_FINISHED ();
END_IF
END_METHOD

METHOD PRIVATE T09_TestEventReport
VAR_INPUT
END_VAR
IF (TcUnit.TEST_ORDERED ('T09_TestEventReport')) THEN
(*	Wyslanie zgloszen	*)
	WRITE_PROTECTED_BOOL (Ptr := ADR (GVL_Variable.fbPB1_K1.bSetError2), Value := TRUE);
	GVL_Variable.fbPB1_K1 ();
	AssertEquals_INT (Expected := 1, Actual := GVL.fbLogger.stBuffer.iNumerOfEvents, 					Message := 'T01a - bledna ilosc w kolejce');
	AssertEquals_INT (Expected := 2, Actual := GVL.fbLogger.stmemory.iNumberOfRow,						Message := 'T01b - bledna ilosc zgloszen');
	GVL.fbLogger ();
	AssertEquals_INT (Expected := 0, Actual := GVL.fbLogger.stBuffer.iNumerOfEvents, 					Message := 'T02a - bledna ilosc w kolejce');
	AssertEquals_INT (Expected := 3, Actual := GVL.fbLogger.stmemory.iNumberOfRow,						Message := 'T02b - bledna ilosc zgloszen');
	AssertEquals_INT (Expected := 1, Actual := GVL.fbLogger.stNumberOfReports.iNumberOfActive,			Message := 'T02c - bledna ilosc zgloszen');
	AssertTrue (Condition := GVL.fbLogger.stNumberOfReports.arrActive [E_BaseEvents_Category.Error],	Message := 'T02d - bledny stan');
	AssertFalse (Condition := GVL.fbLogger.stNumberOfReports.arrActive [E_BaseEvents_Category.Alarm],	Message := 'T02e - bledny stan');
	AssertTrue (Condition := GVL.fbLogger.stNumberOfReports.bIsActive,									Message := 'T02f - bledny stan');
	AssertEquals_INT (Expected := 3, Actual := GVL.fbLogger.stNumberOfReports.iTotalNumer,				Message := 'T02g - bledna ilosc zgloszen');
	AssertEquals_UINT (Expected := 2, Actual := GVL.fbLogger.stMemory.arrRow [1].uiIDItem,				Message := 'T02h - 1 - bledne ID elementu');
	AssertEquals_UINT (Expected := 9, Actual := GVL.fbLogger.stMemory.arrRow [1].uiIDEvent,				Message := 'T02i - 2 - bledne ID zgloszenia');
	AssertEquals_UINT (Expected := 2, Actual := GVL.fbLogger.stMemory.arrRow [2].uiIDItem,				Message := 'T02j - 1 - bledne ID elementu');
	AssertEquals_UINT (Expected := 7, Actual := GVL.fbLogger.stMemory.arrRow [2].uiIDEvent,				Message := 'T02k - 2 - bledne ID zgloszenia');
	AssertEquals_UINT (Expected := 2, Actual := GVL.fbLogger.stMemory.arrRow [3].uiIDItem,				Message := 'T02l - 3 - bledne ID elementu');
	AssertEquals_UINT (Expected := 7, Actual := GVL.fbLogger.stMemory.arrRow [3].uiIDEvent,				Message := 'T02m - 4 - bledne ID zgloszenia');
(*	Wyslanie zgloszen zamnięcie bez potwierdzenia nic sie nie powinno stac*)
	WRITE_PROTECTED_BOOL (Ptr := ADR (GVL_Variable.fbPB1_K1.bResetError2), Value := TRUE);
	GVL_Variable.fbPB1_K1 ();
	AssertEquals_INT (Expected := 1, Actual := GVL.fbLogger.stBuffer.iNumerOfEvents, 					Message := 'T03a - bledna ilosc w kolejce');
	AssertEquals_INT (Expected := 3, Actual := GVL.fbLogger.stmemory.iNumberOfRow,						Message := 'T03b - bledna ilosc zgloszen');
	GVL.fbLogger ();
	AssertEquals_INT (Expected := 0, Actual := GVL.fbLogger.stBuffer.iNumerOfEvents, 					Message := 'T04a - bledna ilosc w kolejce');
	AssertEquals_INT (Expected := 3, Actual := GVL.fbLogger.stmemory.iNumberOfRow,						Message := 'T04b - bledna ilosc zgloszen');
	AssertEquals_INT (Expected := 1, Actual := GVL.fbLogger.stNumberOfReports.iNumberOfActive,			Message := 'T04c - bledna ilosc zgloszen');
	AssertTrue (Condition := GVL.fbLogger.stNumberOfReports.arrActive [E_BaseEvents_Category.Error],	Message := 'T04d - bledny stan');
	AssertFalse (Condition := GVL.fbLogger.stNumberOfReports.arrActive [E_BaseEvents_Category.Alarm],	Message := 'T04e - bledny stan');
	AssertTrue (Condition := GVL.fbLogger.stNumberOfReports.bIsActive,									Message := 'T04f - bledny stan');
	AssertEquals_INT (Expected := 3, Actual := GVL.fbLogger.stNumberOfReports.iTotalNumer,				Message := 'T04g - bledna ilosc zgloszen');
	AssertEquals_UINT (Expected := 2, Actual := GVL.fbLogger.stMemory.arrRow [1].uiIDItem,				Message := 'T04h - 1 - bledne ID elementu');
	AssertEquals_UINT (Expected := 9, Actual := GVL.fbLogger.stMemory.arrRow [1].uiIDEvent,				Message := 'T04i - 2 - bledne ID zgloszenia');
	AssertEquals_UINT (Expected := 2, Actual := GVL.fbLogger.stMemory.arrRow [2].uiIDItem,				Message := 'T04j - 1 - bledne ID elementu');
	AssertEquals_UINT (Expected := 7, Actual := GVL.fbLogger.stMemory.arrRow [2].uiIDEvent,				Message := 'T04k - 2 - bledne ID zgloszenia');
	AssertEquals_UINT (Expected := 2, Actual := GVL.fbLogger.stMemory.arrRow [3].uiIDItem,				Message := 'T04l - 3 - bledne ID elementu');
	AssertEquals_UINT (Expected := 7, Actual := GVL.fbLogger.stMemory.arrRow [3].uiIDEvent,				Message := 'T04m - 4 - bledne ID zgloszenia');
(*	wysłanie potwierdzenia 	*)
	WRITE_PROTECTED_BOOL (Ptr := ADR (GVL_Variable.fbPB1_K1.bAckError2), Value := TRUE);
	GVL_Variable.fbPB1_K1 ();
	AssertEquals_INT (Expected := 1, Actual := GVL.fbLogger.stBuffer.iNumerOfEvents, 					Message := 'T05a - bledna ilosc w kolejce');
	AssertEquals_INT (Expected := 3, Actual := GVL.fbLogger.stmemory.iNumberOfRow,						Message := 'T05b - bledna ilosc zgloszen');
	GVL.fbLogger ();
	AssertEquals_INT (Expected := 0, Actual := GVL.fbLogger.stBuffer.iNumerOfEvents, 					Message := 'T06a - bledna ilosc w kolejce');
	AssertEquals_INT (Expected := 3, Actual := GVL.fbLogger.stmemory.iNumberOfRow,						Message := 'T06b - bledna ilosc zgloszen');
	AssertEquals_INT (Expected := 1, Actual := GVL.fbLogger.stNumberOfReports.iNumberOfActive,			Message := 'T06c - bledna ilosc zgloszen');
	AssertTrue (Condition := GVL.fbLogger.stNumberOfReports.arrActive [E_BaseEvents_Category.Error],	Message := 'T06d - bledny stan');
	AssertFalse (Condition := GVL.fbLogger.stNumberOfReports.arrActive [E_BaseEvents_Category.Alarm],	Message := 'T06e - bledny stan');
	AssertTrue (Condition := GVL.fbLogger.stNumberOfReports.bIsActive,									Message := 'T06f - bledny stan');
	AssertEquals_INT (Expected := 3, Actual := GVL.fbLogger.stNumberOfReports.iTotalNumer,				Message := 'T06g - bledna ilosc zgloszen');
	AssertEquals_UINT (Expected := 2, Actual := GVL.fbLogger.stMemory.arrRow [1].uiIDItem,				Message := 'T06h - 1 - bledne ID elementu');
	AssertEquals_UINT (Expected := 9, Actual := GVL.fbLogger.stMemory.arrRow [1].uiIDEvent,				Message := 'T06i - 2 - bledne ID zgloszenia');
	AssertEquals_UINT (Expected := 2, Actual := GVL.fbLogger.stMemory.arrRow [2].uiIDItem,				Message := 'T06j - 1 - bledne ID elementu');
	AssertEquals_UINT (Expected := 7, Actual := GVL.fbLogger.stMemory.arrRow [2].uiIDEvent,				Message := 'T06k - 2 - bledne ID zgloszenia');
	AssertEquals_UINT (Expected := 2, Actual := GVL.fbLogger.stMemory.arrRow [3].uiIDItem,				Message := 'T06l - 3 - bledne ID elementu');
	AssertEquals_UINT (Expected := 7, Actual := GVL.fbLogger.stMemory.arrRow [3].uiIDEvent,				Message := 'T06m - 4 - bledne ID zgloszenia');
(*	Wyslanie zgloszen zamnięcie *)
	WRITE_PROTECTED_BOOL (Ptr := ADR (GVL_Variable.fbPB1_K1.bReseterror2), Value := TRUE);
	GVL_Variable.fbPB1_K1 ();
	AssertEquals_INT (Expected := 1, Actual := GVL.fbLogger.stBuffer.iNumerOfEvents, 					Message := 'T07a - bledna ilosc w kolejce');
	AssertEquals_INT (Expected := 3, Actual := GVL.fbLogger.stmemory.iNumberOfRow,						Message := 'T07b - bledna ilosc zgloszen');
	GVL.fbLogger ();
	AssertEquals_INT (Expected := 0, Actual := GVL.fbLogger.stBuffer.iNumerOfEvents, 					Message := 'T08a - bledna ilosc w kolejce');
	AssertEquals_INT (Expected := 3, Actual := GVL.fbLogger.stmemory.iNumberOfRow,						Message := 'T08b - bledna ilosc zgloszen');
	AssertEquals_INT (Expected := 0, Actual := GVL.fbLogger.stNumberOfReports.iNumberOfActive,			Message := 'T08c - bledna ilosc zgloszen');
	AssertFalse (Condition := GVL.fbLogger.stNumberOfReports.arrActive [E_BaseEvents_Category.Error],	Message := 'T08d - bledny stan');
	AssertFalse (Condition := GVL.fbLogger.stNumberOfReports.arrActive [E_BaseEvents_Category.Alarm],	Message := 'T08e - bledny stan');
	AssertFalse (Condition := GVL.fbLogger.stNumberOfReports.bIsActive,									Message := 'T08f - bledny stan');
	AssertEquals_INT (Expected := 3, Actual := GVL.fbLogger.stNumberOfReports.iTotalNumer,				Message := 'T08g - bledna ilosc zgloszen');
	AssertEquals_UINT (Expected := 2, Actual := GVL.fbLogger.stMemory.arrRow [1].uiIDItem,				Message := 'T08h - 1 - bledne ID elementu');
	AssertEquals_UINT (Expected := 9, Actual := GVL.fbLogger.stMemory.arrRow [1].uiIDEvent,				Message := 'T08i - 2 - bledne ID zgloszenia');
	AssertEquals_UINT (Expected := 2, Actual := GVL.fbLogger.stMemory.arrRow [2].uiIDItem,				Message := 'T08j - 1 - bledne ID elementu');
	AssertEquals_UINT (Expected := 7, Actual := GVL.fbLogger.stMemory.arrRow [2].uiIDEvent,				Message := 'T08k - 2 - bledne ID zgloszenia');
	AssertEquals_UINT (Expected := 2, Actual := GVL.fbLogger.stMemory.arrRow [3].uiIDItem,				Message := 'T08l - 3 - bledne ID elementu');
	AssertEquals_UINT (Expected := 7, Actual := GVL.fbLogger.stMemory.arrRow [3].uiIDEvent,				Message := 'T08m - 4 - bledne ID zgloszenia');
	
	TcUnit.TEST_FINISHED ();
END_IF
END_METHOD

METHOD PRIVATE T10_PreparetableEventsForTesting
VAR_INPUT
END_VAR
IF (TcUnit.TEST_ORDERED ('T10_PreparetableEventsForTesting')) THEN
	WRITE_PROTECTED_BOOL (Ptr := ADR (GVL_Variable.fbPB1_Wyk1_K1.bSetAlarm2), Value := TRUE);
	GVL_Variable.fbPB1_Wyk1_K1 ();
	WRITE_PROTECTED_BOOL (Ptr := ADR (GVL_Variable.fbPB1_K1.bSetAlarm2), Value := TRUE);
	GVL_Variable.fbPB1_K1 ();
	WRITE_PROTECTED_BOOL (Ptr := ADR (GVL_Variable.fbPB1_ZL1_Wyk1_K1.bSetError2), Value := TRUE);
	GVL_Variable.fbPB1_ZL1_Wyk1_K1 ();
	GVL.fbLogger ();
	WRITE_PROTECTED_BOOL (Ptr := ADR (GVL_Variable.fbPB1_K1.bSetError2), Value := TRUE);
	GVL_Variable.fbPB1_K1 ();
	WRITE_PROTECTED_BOOL (Ptr := ADR (GVL_Variable.fbPB1_K1.bSetError4), Value := TRUE);
	GVL_Variable.fbPB1_K1 ();
	WRITE_PROTECTED_BOOL (Ptr := ADR (GVL_Variable.fbPB1_Wyk2_K1.bSetAlarm), Value := TRUE);
	GVL_Variable.fbPB1_Wyk2_K1 ();
	GVL.fbLogger ();
	WRITE_PROTECTED_BOOL (Ptr := ADR (GVL_Variable.fbPB1_K1.bResetAlarm2), Value := TRUE);
	GVL_Variable.fbPB1_K1 ();
	WRITE_PROTECTED_BOOL (Ptr := ADR (GVL_Variable.fbPB1_Wyk1_K1.bResetAlarm2), Value := TRUE);
	GVL_Variable.fbPB1_Wyk1_K1 ();
	WRITE_PROTECTED_BOOL (Ptr := ADR (GVL_Variable.fbPB1_K1.bSetError1), Value := TRUE);
	GVL_Variable.fbPB1_K1 ();
	GVL.fbLogger ();
	TcUnit.TEST_FINISHED ();
END_IF
END_METHOD

METHOD PRIVATE T11_TestGenerateListEvent
VAR_INPUT
END_VAR
IF (TcUnit.TEST_ORDERED ('T11_TestGenerateListEvent')) THEN
	GVL_VariableHMI.fbPB1_K1_HMI.GetYourEventTable ();
	AssertEquals_INT (Expected := 7, Actual := GVL.fbLogger.arrNumberOfReportsForItem [2].iTotalNumer, Message := 'T01 - bledna ilosc zgloszen');
	AssertEquals_INT (Expected := 3, Actual := GVL.fbLogger.arrNumberOfReportsForItem [2].iNumberOfActive, Message := 'T02 - bledna ilosc zgloszen aktywnych');
	AssertTrue (Condition := GVL.fbLogger.arrNumberOfReportsForItem [2].bIsActive, Message := 'T03 - bledny stan aktywnosci');
	AssertTrue (Condition := GVL.fbLogger.arrNumberOfReportsForItem [2].bIsActiveWithConfirmation, Message := 'T04 - bledny stan do potwierdzenia');
	
	AssertEquals_INT (Expected := 3, Actual := GVL.fbLogger.arrNumberOfReportsForItem [2].arrNumberOfActive [1], Message := 'T05 - bledna ilosc zgloszen');
	AssertEquals_INT (Expected := 0, Actual := GVL.fbLogger.arrNumberOfReportsForItem [2].arrNumberOfActive [2], Message := 'T06 - bledna ilosc zgloszen');
	AssertTrue (Condition := GVL.fbLogger.arrNumberOfReportsForItem [2].arrActive [1], Message := 'T07 - bledny stan');
	AssertFalse (Condition := GVL.fbLogger.arrNumberOfReportsForItem [2].arrActive [2], Message := 'T08 - bledny stan');
	
	AssertEquals_INT (Expected := 7, Actual := GVL_VariableHMI.fbPB1_K1_HMI.refstBaseLoggerElementDataHMI.stListOfEventsToDisplay.iNumberOfRow , Message := 'T10 - bledna ilosc do wyswietlenia');
	AssertEquals_UINT (Expected := 8, Actual := GVL_VariableHMI.fbPB1_K1_HMI.refstBaseLoggerElementDataHMI.stListOfEventsToDisplay.arrToDisplay [1].uiIDEvent , Message := 'T10 - [01] - Bledny ID zdarzenia');
	AssertEquals_UINT (Expected := 12, Actual := GVL_VariableHMI.fbPB1_K1_HMI.refstBaseLoggerElementDataHMI.stListOfEventsToDisplay.arrToDisplay [2].uiIDEvent , Message := 'T10 - [02] - Bledny ID zdarzenia');
	AssertEquals_UINT (Expected := 9, Actual := GVL_VariableHMI.fbPB1_K1_HMI.refstBaseLoggerElementDataHMI.stListOfEventsToDisplay.arrToDisplay [3].uiIDEvent , Message := 'T10 - [03] - Bledny ID zdarzenia');
	AssertEquals_UINT (Expected := 10, Actual := GVL_VariableHMI.fbPB1_K1_HMI.refstBaseLoggerElementDataHMI.stListOfEventsToDisplay.arrToDisplay [4].uiIDEvent , Message := 'T10 - [04] - Bledny ID zdarzenia');
	AssertEquals_UINT (Expected := 9, Actual := GVL_VariableHMI.fbPB1_K1_HMI.refstBaseLoggerElementDataHMI.stListOfEventsToDisplay.arrToDisplay [5].uiIDEvent , Message := 'T10 - [05] - Bledny ID zdarzenia');
	AssertEquals_UINT (Expected := 7, Actual := GVL_VariableHMI.fbPB1_K1_HMI.refstBaseLoggerElementDataHMI.stListOfEventsToDisplay.arrToDisplay [6].uiIDEvent , Message := 'T10 - [06] - Bledny ID zdarzenia');
	AssertEquals_UINT (Expected := 7, Actual := GVL_VariableHMI.fbPB1_K1_HMI.refstBaseLoggerElementDataHMI.stListOfEventsToDisplay.arrToDisplay [7].uiIDEvent , Message := 'T10 - [07] - Bledny ID zdarzenia');
	
//tylko aktywne	
	GVL.stTopElementData.stComponent1.stBaseLoggerElement.stFilter.bActive	:= TRUE;
	GVL_VariableHMI.fbPB1_K1_HMI.GetYourEventTable ();
	AssertEquals_INT (Expected := 3, Actual := GVL_VariableHMI.fbPB1_K1_HMI.refstBaseLoggerElementDataHMI.stListOfEventsToDisplay.iNumberOfRow , Message := 'T11 - bledna ilosc do wyswietlenia');
	AssertEquals_UINT (Expected := 8, Actual := GVL_VariableHMI.fbPB1_K1_HMI.refstBaseLoggerElementDataHMI.stListOfEventsToDisplay.arrToDisplay [1].uiIDEvent , Message := 'T11 - [01] - Bledny ID zdarzenia');
	AssertEquals_UINT (Expected := 12, Actual := GVL_VariableHMI.fbPB1_K1_HMI.refstBaseLoggerElementDataHMI.stListOfEventsToDisplay.arrToDisplay [2].uiIDEvent , Message := 'T11 - [02] - Bledny ID zdarzenia');
	AssertEquals_UINT (Expected := 9, Actual := GVL_VariableHMI.fbPB1_K1_HMI.refstBaseLoggerElementDataHMI.stListOfEventsToDisplay.arrToDisplay [3].uiIDEvent , Message := 'T11 - [03] - Bledny ID zdarzenia');
	
//tylko nie aktywne	
	GVL.stTopElementData.stComponent1.stBaseLoggerElement.stFilter.bActive	:= FALSE;
	GVL.stTopElementData.stComponent1.stBaseLoggerElement.stFilter.bNotActive	:= TRUE;	
	GVL_VariableHMI.fbPB1_K1_HMI.GetYourEventTable ();
	AssertEquals_INT (Expected := 4, Actual := GVL_VariableHMI.fbPB1_K1_HMI.refstBaseLoggerElementDataHMI.stListOfEventsToDisplay.iNumberOfRow , Message := 'T12 - bledna ilosc do wyswietlenia');
	AssertEquals_UINT (Expected := 10, Actual := GVL_VariableHMI.fbPB1_K1_HMI.refstBaseLoggerElementDataHMI.stListOfEventsToDisplay.arrToDisplay [1].uiIDEvent , Message := 'T12 - [01] - Bledny ID zdarzenia');
	AssertEquals_UINT (Expected := 9, Actual := GVL_VariableHMI.fbPB1_K1_HMI.refstBaseLoggerElementDataHMI.stListOfEventsToDisplay.arrToDisplay [2].uiIDEvent , Message := 'T12 - [02] - Bledny ID zdarzenia');
	AssertEquals_UINT (Expected := 7, Actual := GVL_VariableHMI.fbPB1_K1_HMI.refstBaseLoggerElementDataHMI.stListOfEventsToDisplay.arrToDisplay [3].uiIDEvent , Message := 'T12 - [03] - Bledny ID zdarzenia');
	AssertEquals_UINT (Expected := 7, Actual := GVL_VariableHMI.fbPB1_K1_HMI.refstBaseLoggerElementDataHMI.stListOfEventsToDisplay.arrToDisplay [4].uiIDEvent , Message := 'T12 - [04] - Bledny ID zdarzenia');

	GVL.stTopElementData.stComponent1.stBaseLoggerElement.stFilter.bNotActive	:= FALSE;	
	GVL_VariableHMI.fbPB1_K1_HMI.GetYourEventTable ();
	AssertEquals_INT (Expected := 7, Actual := GVL_VariableHMI.fbPB1_K1_HMI.refstBaseLoggerElementDataHMI.stListOfEventsToDisplay.iNumberOfRow , Message := 'T13 - bledna ilosc do wyswietlenia');
	AssertEquals_UINT (Expected := 8, Actual := GVL_VariableHMI.fbPB1_K1_HMI.refstBaseLoggerElementDataHMI.stListOfEventsToDisplay.arrToDisplay [1].uiIDEvent , Message := 'T13 - [01] - Bledny ID zdarzenia');
	AssertEquals_UINT (Expected := 12, Actual := GVL_VariableHMI.fbPB1_K1_HMI.refstBaseLoggerElementDataHMI.stListOfEventsToDisplay.arrToDisplay [2].uiIDEvent , Message := 'T13 - [02] - Bledny ID zdarzenia');
	AssertEquals_UINT (Expected := 9, Actual := GVL_VariableHMI.fbPB1_K1_HMI.refstBaseLoggerElementDataHMI.stListOfEventsToDisplay.arrToDisplay [3].uiIDEvent , Message := 'T13 - [03] - Bledny ID zdarzenia');
	AssertEquals_UINT (Expected := 10, Actual := GVL_VariableHMI.fbPB1_K1_HMI.refstBaseLoggerElementDataHMI.stListOfEventsToDisplay.arrToDisplay [4].uiIDEvent , Message := 'T13 - [04] - Bledny ID zdarzenia');
	AssertEquals_UINT (Expected := 9, Actual := GVL_VariableHMI.fbPB1_K1_HMI.refstBaseLoggerElementDataHMI.stListOfEventsToDisplay.arrToDisplay [5].uiIDEvent , Message := 'T13 - [05] - Bledny ID zdarzenia');
	AssertEquals_UINT (Expected := 7, Actual := GVL_VariableHMI.fbPB1_K1_HMI.refstBaseLoggerElementDataHMI.stListOfEventsToDisplay.arrToDisplay [6].uiIDEvent , Message := 'T13 - [06] - Bledny ID zdarzenia');
	AssertEquals_UINT (Expected := 7, Actual := GVL_VariableHMI.fbPB1_K1_HMI.refstBaseLoggerElementDataHMI.stListOfEventsToDisplay.arrToDisplay [7].uiIDEvent , Message := 'T13 - [07] - Bledny ID zdarzenia');

	
	TcUnit.TEST_FINISHED ();
END_IF
END_METHOD

METHOD PROTECTED T12_TestPower
VAR_INST
	iStep				: INT;
END_VAR
IF (TcUnit.TEST_ORDERED ('T12_TestPower')) THEN
	CASE iStep OF
	0	:
		AssertFalse (Condition := GVL.fbSS1.GetFlag (), Message := 'S00 - T01 - Bledny stan');
		AssertFalse (Condition := GVL.fbSTO.GetFlag (), Message := 'S00 - T02 - Bledny stan');
		GVL_Variable.fbPB1_Wyk1.PowerTurnOn ();
		iStep		:= iStep + 10;
	10	:
		GVL_Variable.fbPB1_Wyk1.ExecuteEveryCycle_Test ();
		GVL_Variable.fbPB1_Wyk1.ExecuteEveryCycle_Operation ();
		AssertFalse (Condition := GVL_Variable.fbPB1_Wyk1.stEvents.arrState [1], 				Message := 'S10 - T01 - bledny stan bledu SS1');
		AssertFalse (Condition := GVL_Variable.fbPB1_Wyk1.stEvents.arrState [2], 				Message := 'S10 - T02 - bledny stan bledu STO');
		AssertTrue (Condition := GVL_Variable.fbPB1_Wyk1.stPower.cmdTurnOn.IsBusy (), 			Message := 'S10 - T03 - bledny stan trwa');
		AssertTrue (Condition := GVL_Variable.fbPB1_Wyk1.stPower.cmdTurnOn.IsFirstCycle (), 	Message := 'S10 - T05 - bledny pierwszy cykl');
		AssertFalse (Condition := GVL_Variable.fbPB1_Wyk1.stPower.cmdTurnOn.IsLastCycle (), 	Message := 'S10 - T06 - bledny ostatni cykl');
		AssertFalse (Condition := GVL_Variable.fbPB1_Wyk1.PowerGetStatus (), 					Message := 'S10 - T04 - bledny status');
		
		iStep		:= iStep + 10;
	20	:
		GVL_Variable.fbPB1_Wyk1.ExecuteEveryCycle_Test ();
		GVL_Variable.fbPB1_Wyk1.ExecuteEveryCycle_Operation ();
		AssertTrue (Condition := GVL_Variable.fbPB1_Wyk1.stEvents.arrState [1], 				Message := 'T20 - 01 - bledny stan bledu SS1');
		AssertTrue (Condition := GVL_Variable.fbPB1_Wyk1.stEvents.arrState [2], 				Message := 'T20 - 02 - bledny stan bledu STO');
		AssertFalse (Condition := GVL_Variable.fbPB1_Wyk1.stPower.cmdTurnOn.IsBusy (),		 	Message := 'T20 - 03 - bledny stan trwa');
		AssertFalse (Condition := GVL_Variable.fbPB1_Wyk1.stPower.cmdTurnOn.IsFirstCycle (),	Message := 'T20 - 05 - bledny pierwszy cykl');
		AssertFalse (Condition := GVL_Variable.fbPB1_Wyk1.stpower.cmdTurnOn.IsLastCycle (), 	Message := 'T20 - 06 - bledny ostatni cykl');
		AssertFalse (Condition := GVL_Variable.fbPB1_Wyk1.PowerGetStatus (), 					Message := 'T20 - 04 - bledny status');
		GVL.fbSS1.SetFlag (bState := TRUE);
		GVL.fbSTO.SetFlag (bState := TRUE);
		iStep			:= iStep + 10;
	30	:
		GVL_Variable.fbPB1_Wyk1.ExecuteEveryCycle_Test ();
		GVL_Variable.fbPB1_Wyk1.ExecuteEveryCycle_Operation ();
		iStep			:= iStep + 10;
	40	:
		GVL_Variable.fbPB1_Wyk1.PowerTurnOn ();
		iStep			:= iStep + 10;
	50	:
		GVL_Variable.fbPB1_Wyk1.ExecuteEveryCycle_Test ();
		GVL_Variable.fbPB1_Wyk1.ExecuteEveryCycle_Operation ();
		AssertTrue (Condition := GVL_Variable.fbPB1_Wyk1.stEvents.arrState [1], 						Message := 'T50 - 01 - bledny stan bledu SS1');
		AssertTrue (Condition := GVL_Variable.fbPB1_Wyk1.stEvents.arrState [2],				 			Message := 'T50 - 02 - bledny stan bledu STO');
		AssertTrue (Condition := GVL_Variable.fbPB1_Wyk1.stPower.cmdTurnOn.IsBusy (),				 	Message := 'T50 - 03 - bledny stan trwa');
		AssertFalse (Condition := GVL_Variable.fbPB1_Wyk1.PowerGetStatus (),			 				Message := 'T50 - 04 - bledny status');
		iStep			:= iStep + 10;
	60	:
		GVL_Variable.fbPB1_Wyk1.ExecuteEveryCycle_Test ();
		GVL_Variable.fbPB1_Wyk1.ExecuteEveryCycle_Operation ();
		AssertFalse (Condition := GVL_Variable.fbPB1_Wyk1.stEvents.arrState [1], 						Message := 'T60 - 01 - bledny stan bledu SS1');
		AssertFalse (Condition := GVL_Variable.fbPB1_Wyk1.stEvents.arrState [2], 						Message := 'T60 - 02 - bledny stan bledu STO');
		AssertTrue (Condition := GVL_Variable.fbPB1_Wyk1.stPower.cmdTurnOn.IsBusy (),				 	Message := 'T60 - 03 - bledny stan trwa');
		AssertTrue (Condition := GVL_Variable.fbPB1_Wyk1.PowerGetStatus (), 							Message := 'T60 - 04 - bledny status');
		iStep			:= iStep + 10;
	70	:
		GVL_Variable.fbPB1_Wyk1.ExecuteEveryCycle_Test ();
		GVL_Variable.fbPB1_Wyk1.ExecuteEveryCycle_Operation ();
		AssertFalse (Condition := GVL_Variable.fbPB1_Wyk1.stpower.cmdTurnOn.IsBusy (), 				Message := 'T70 - 01 - bledny stan trwa');
		AssertTrue (Condition := GVL_Variable.fbPB1_Wyk1.PowerGetStatus(),			 					Message := 'T70 - 02 - bledny status');
		iStep			:= iStep + 10;
	80	:
		GVL_Variable.fbPB1_Wyk1.ExecuteEveryCycle_Test ();
		GVL_Variable.fbPB1_Wyk1.ExecuteEveryCycle_Operation ();
		iStep			:= iStep + 10;
	90	:
		GVL_Variable.fbPB1_Wyk1.PowerTurnOff ();
		iStep			:= iStep + 10;
	100	:
		GVL_Variable.fbPB1_Wyk1.ExecuteEveryCycle_Test ();
		GVL_Variable.fbPB1_Wyk1.ExecuteEveryCycle_Operation ();
		AssertTrue (Condition := GVL_Variable.fbPB1_Wyk1.stPower.cmdTurnOff.IsBusy (), 	Message := 'T100 - 03 - bledny stan trwa');
		AssertTrue (Condition := GVL_Variable.fbPB1_Wyk1.PowerGetStatus (), 				Message := 'T100 - 04 - bledny status');
		iStep			:= iStep + 10;
	110	:
		GVL_Variable.fbPB1_Wyk1.ExecuteEveryCycle_Test ();
		GVL_Variable.fbPB1_Wyk1.ExecuteEveryCycle_Operation ();
		AssertTrue (Condition := GVL_variable.fbPB1_Wyk1.stPower.cmdTurnOff.IsBusy (), 	Message := 'T110 - 03 - bledny stan trwa');
		AssertFalse (Condition := GVL_Variable.fbPB1_Wyk1.PowerGetStatus (), 					Message := 'T110 - 04 - bledny status');
		iStep			:= iStep + 10;
	120	:
		GVL_Variable.fbPB1_Wyk1.ExecuteEveryCycle_Test ();
		GVL_Variable.fbPB1_Wyk1.ExecuteEveryCycle_Operation ();
		AssertFalse (Condition := GVL_Variable.fbPB1_Wyk1.stPower.cmdTurnOff.IsBusy (), 	Message := 'T120 - 01 - bledny stan trwa');
		AssertFalse (Condition := GVL_Variable.fbPB1_Wyk1.PowerGetStatus (), 					Message := 'T120 - 02 - bledny status');
		


		iStep		:= 1000;
	1000	:
		TcUnit.TEST_FINISHED ();
	END_CASE
END_IF
END_METHOD

